	J1=     0.000 deg,	J2=   180.000 deg
};
P[172]{
   GP1:
	UF : 1, UT : 1,		CONFIG : 'N U T, 0, 0, 0',
	X =  2112.025  mm,	Y =   402.590  mm,	Z =  1192.449  mm,
	W =      .016 deg,	P =     -.045 deg,	R =   -23.885 deg
   GP2:
	UF : 1, UT : 1,
	J1=   135.000 deg,	J2=     0.000 deg
};
P[173]{
   GP1:
	UF : 1, UT : 1,		CONFIG : 'N U T, 0, 0, 0',
	X =  2111.810  mm,	Y =    14.647  mm,	Z =  1192.450  mm,
	W =      .016 deg,	P =     -.045 deg,	R =   -23.885 deg
   GP2:
	UF : 1, UT : 1,
	J1=   135.000 deg,	J2=     0.000 deg
};
P[174]{
   GP1:
	UF : 1, UT : 1,		CONFIG : 'N U T, 0, 0, 0',
	X =  1543.269  mm,	Y =  -478.741  mm,	Z =    98.416  mm,
	W =   -16.138 deg,	P =    42.751 deg,	R =   168.873 deg
   GP2:
	UF : 1, UT : 1,
	J1=     0.000 deg,	J2=   180.000 deg
};
P[175]{
   GP1:
	UF : 1, UT : 1,		CONFIG : 'N U T, 0, 0, 0',
	X =  1494.684  mm,	Y =    -9.285  mm,	Z =   211.201  mm,
	W =    -1.993 deg,	P =    44.965 deg,	R =   177.180 deg
   GP2:
	UF : 1, UT : 1,
	J1=     0.000 deg,	J2=   180.000 deg
};
P[176]{
   GP1:
	UF : 1, UT : 1,		CONFIG : 'N U T, 0, 0, 0',
	X =  2128.997  mm,	Y =  -645.877  mm,	Z =  1179.040  mm,
	W =     -.110 deg,	P =     -.657 deg,	R =   -23.879 deg
   GP2:
	UF : 1, UT : 1,
	J1=   135.000 deg,	J2=     0.000 deg
};
P[177]{
   GP1:
	UF : 1, UT : 1,		CONFIG : 'N U T, 0, 0, 0',
	X =  2128.776  mm,	Y =  -455.457  mm,	Z =  1177.054  mm,
	W =     -.064 deg,	P =    -1.106 deg,	R =   -23.872 deg
   GP2:
	UF : 1, UT : 1,
	J1=   135.000 deg,	J2=     0.000 deg
};
P[178]{
   GP1:
	UF : 1, UT : 1,		CONFIG : 'N U T, 0, 0, 0',
	X =  1534.968  mm,	Y =  -398.034  mm,	Z =    84.062  mm,
	W =     -.043 deg,	P =    44.368 deg,	R =   176.047 deg
   GP2:
	UF : 1, UT : 1,
	J1=     0.000 deg,	J2=   180.000 deg
};
P[179]{
   GP1:
	UF : 1, UT : 1,		CONFIG : 'N U T, 0, 0, 0',
	X =  1493.431  mm,	Y =   363.490  mm,	Z =   189.000  mm,
	W =   -16.664 deg,	P =    42.430 deg,	R =   156.075 deg
   GP2:
	UF : 1, UT : 1,
	J1=     0.000 deg,	J2=   180.000 deg
};
P[180]{
   GP1:
	UF : 1, UT : 1,		CONFIG : 'N U T, 0, 0, 0',
	X =  2129.638  mm,	Y =  -446.131  mm,	Z =  1180.944  mm,
	W =     3.415 deg,	P =     -.816 deg,	R =   -23.974 deg
   GP2:
	UF : 1, UT : 1,
	J1=   135.000 deg,	J2=     0.000 deg
};
P[181]{
   GP1:
	UF : 1, UT : 1,		CONFIG : 'N U T, 0, 0, 0',
	X =  2353.698  mm,	Y =   399.991  mm,	Z =   291.072  mm,
	W =    43.149 deg,	P =    14.488 deg,	R =   -37.828 deg
   GP2:
	UF : 1, UT : 1,
	J1=      .000 deg,	J2=   180.000 deg
};
P[182]{
   GP1:
	UF : 1, UT : 1,		CONFIG : 'N U T, 0, 0, 0',
	X =  1481.802  mm,	Y =    -4.268  mm,	Z =   197.574  mm,
	W =    -1.993 deg,	P =    44.965 deg,	R =   177.180 deg
   GP2:
	UF : 1, UT : 1,
	J1=     0.000 deg,	J2=   180.000 deg
};
P[183]{
   GP1:
	UF : 1, UT : 1,		CONFIG : 'N U T, 0, 0, 0',
	X =  1481.802  mm,	Y =   612.875  mm,	Z =   197.574  mm,
	W =   -40.373 deg,	P =    21.850 deg,	R =   111.598 deg
   GP2:
	UF : 1, UT : 1,
	J1=     0.000 deg,	J2=   180.000 deg
};
P[184]{
   GP1:
	UF : 1, UT : 1,		CONFIG : 'N U T, 0, 0, 0',
	X =  2345.067  mm,	Y =   409.224  mm,	Z =   281.500  mm,
	W =    43.108 deg,	P =    14.444 deg,	R =   -17.326 deg
   GP2:
	UF : 1, UT : 1,
	J1=     0.000 deg,	J2=   180.000 deg
};
P[185]{
   GP1:
	UF : 1, UT : 1,		CONFIG : 'N U T, 0, 0, 0',
	X =  2306.742  mm,	Y =   406.911  mm,	Z =   281.490  mm,
	W =    43.110 deg,	P =    14.442 deg,	R =   -17.330 deg
   GP2:
	UF : 1, UT : 1,
	J1=     0.000 deg,	J2=   180.000 deg
};
P[186]{
   GP1:
	UF : 1, UT : 1,		CONFIG : 'N U T, 0, 0, -1',
	X =  1406.501  mm,	Y =   510.995  mm,	Z =   296.764  mm,
	W =   -40.802 deg,	P =    20.911 deg,	R =   112.463 deg
   GP2:
	UF : 1, UT : 1,
	J1=     0.000 deg,	J2=   180.000 deg
};
P[187]{
   GP1:
	UF : 1, UT : 1,		CONFIG : 'N U T, 0, 0, 0',
	X =  1226.008  mm,	Y =   -21.205  mm,	Z =   297.416  mm,
	W =      .340 deg,	P =    45.409 deg,	R =    12.184 deg
   GP2:
	UF : 1, UT : 1,
	J1=     0.000 deg,	J2=   180.000 deg
};
P[188]{
   GP1:
	UF : 1, UT : 1,		CONFIG : 'N U T, 0, 0, 0',
	X =  2197.405  mm,	Y =   -25.809  mm,	Z =  -200.004  mm,
	W =     -.223 deg,	P =     -.454 deg,	R =     -.269 deg
   GP2:
	UF : 1, UT : 1,
	J1=    45.206 deg,	J2=   180.000 deg
};
P[189]{
   GP1:
	UF : 1, UT : 1,		CONFIG : 'N U T, 0, 0, 0',
	X =  2305.896  mm,	Y =   -25.032  mm,	Z =  -270.188  mm,
	W =      .477 deg,	P =    12.556 deg,	R =     -.810 deg
   GP2:
	UF : 1, UT : 1,
	J1=    45.206 deg,	J2=   180.000 deg
};
P[190]{
   GP1:
	UF : 1, UT : 1,		CONFIG : 'N U T, 0, 0, 0',
	X =  2290.712  mm,	Y =   409.911  mm,	Z =   281.500  mm,
	W =    43.107 deg,	P =    14.443 deg,	R =    14.426 deg
   GP2:
	UF : 1, UT : 1,
	J1=     0.000 deg,	J2=   180.000 deg
};
P[191]{
   GP1:
	UF : 1, UT : 1,		CONFIG : 'N U T, 0, 0, 0',
	X =  2361.728  mm,	Y =  -412.684  mm,	Z =   283.675  mm,
	W =   -31.226 deg,	P =   -24.163 deg,	R =    -2.589 deg
   GP2:
	UF : 1, UT : 1,
	J1=     0.000 deg,	J2=   180.000 deg
};
P[192]{
   GP1:
	UF : 1, UT : 1,		CONFIG : 'N U T, 0, 0, 0',
	X =  2327.653  mm,	Y =   -25.077  mm,	Z =  -148.093  mm,
	W =      .476 deg,	P =    12.559 deg,	R =     -.810 deg
   GP2:
	UF : 1, UT : 1,
	J1=    45.206 deg,	J2=   180.000 deg
};
P[193]{
   GP1:
	UF : 1, UT : 1,		CONFIG : 'N U T, 0, 0, 0',
	X =  1727.799  mm,	Y =   -46.845  mm,	Z =   458.542  mm,
	W =     2.935 deg,	P =   -34.514 deg,	R =   -11.373 deg
   GP2:
	UF : 1, UT : 1,
	J1=     0.000 deg,	J2=   180.000 deg
};
P[194]{
   GP1:
	UF : 1, UT : 1,		CONFIG : 'N U T, 0, 0, 0',
	X =  2344.238  mm,	Y =  -414.136  mm,	Z =   281.331  mm,
	W =   -33.506 deg,	P =   -24.171 deg,	R =   -30.020 deg
   GP2:
	UF : 1, UT : 1,
	J1=     0.000 deg,	J2=   180.000 deg
};
P[195]{
   GP1:
	UF : 1, UT : 1,		CONFIG : 'N U T, 0, 0, 0',
	X =  2303.808  mm,	Y =  -413.308  mm,	Z =   281.330  mm,
	W =   -33.506 deg,	P =   -24.171 deg,	R =   -30.020 deg
   GP2:
	UF : 1, UT : 1,
	J1=     0.000 deg,	J2=   180.000 deg
};
P[196]{
   GP1:
	UF : 1, UT : 1,		CONFIG : 'N U T, 0, 0, 0',
	X =  1670.118  mm,	Y =  -166.484  mm,	Z =   -15.328  mm,
	W =     1.674 deg,	P =   -29.607 deg,	R =   -12.085 deg
   GP2:
	UF : 1, UT : 1,
	J1=     0.000 deg,	J2=   180.000 deg
};
P[197]{
   GP1:
	UF : 1, UT : 1,		CONFIG : 'N U T, 0, 0, 0',
	X =  2284.901  mm,	Y =  -412.985  mm,	Z =   282.798  mm,
	W =   -33.505 deg,	P =   -24.171 deg,	R =   -60.790 deg
   GP2:
	UF : 1, UT : 1,
	J1=     0.000 deg,	J2=   180.000 deg
};
P[198]{
   GP1:
	UF : 1, UT : 1,		CONFIG : 'N U T, 0, 0, 0',
	X =  2368.954  mm,	Y =  -246.180  mm,	Z =  -185.021  mm,
	W =    35.524 deg,	P =    28.328 deg,	R =  -122.465 deg
   GP2:
	UF : 1, UT : 1,
	J1=      .000 deg,	J2=   180.000 deg
};
P[199]{
   GP1:
	UF : 1, UT : 1,		CONFIG : 'N U T, 0, 0, 0',
	X =  1667.363  mm,	Y =  -120.483  mm,	Z =     2.410  mm,
	W =     6.134 deg,	P =   -28.692 deg,	R =   -14.256 deg
   GP2:
	UF : 1, UT : 1,
	J1=     0.000 deg,	J2=   180.000 deg
};
P[200]{
   GP1:
	UF : 1, UT : 1,		CONFIG : 'N U T, 0, 0, 0',
	X =  1526.901  mm,	Y =   -72.453  mm,	Z =   656.445  mm,
	W =   -14.352 deg,	P =    -5.632 deg,	R =   -30.177 deg
   GP2:
	UF : 1, UT : 1,
	J1=     0.000 deg,	J2=   180.000 deg
};
P[201]{
   GP1:
	UF : 1, UT : 1,		CONFIG : 'N U T, 0, 0, 0',
	X =   918.616  mm,	Y =  -238.769  mm,	Z =   572.023  mm,
	W =    44.545 deg,	P =     7.177 deg,	R =    -7.219 deg
   GP2:
	UF : 1, UT : 1,
	J1=    80.000 deg,	J2=    90.000 deg
};
P[202]{
   GP1:
	UF : 1, UT : 1,		CONFIG : 'N U T, 0, 0, 0',
	X =  1548.492  mm,	Y = -1079.480  mm,	Z =  1677.351  mm,
	W =   -38.101 deg,	P =   -29.846 deg,	R =   -22.090 deg
   GP2:
	UF : 1, UT : 1,
	J1=   180.000 deg,	J2=   -90.000 deg
};
P[203]{
   GP1:
	UF : 1, UT : 1,		CONFIG : 'N U T, 0, 0, 0',
	X =  2472.617  mm,	Y =   -96.769  mm,	Z =    57.023  mm,
	W =    44.545 deg,	P =     7.177 deg,	R =    -7.219 deg
   GP2:
	UF : 1, UT : 1,
	J1=    80.000 deg,	J2=    90.000 deg
};
P[204]{
   GP1:
	UF : 1, UT : 1,		CONFIG : 'N U T, 0, 0, 0',
	X =  2434.636  mm,	Y =    22.422  mm,	Z =     9.532  mm,
	W =    44.545 deg,	P =     7.177 deg,	R =     8.203 deg
   GP2:
	UF : 1, UT : 1,
	J1=    80.000 deg,	J2=    90.000 deg
};
P[205]{
   GP1:
	UF : 1, UT : 1,		CONFIG : 'N U T, 0, 0, 0',
	X =  2368.508  mm,	Y =  -153.263  mm,	Z =  -185.665  mm,
	W =    29.649 deg,	P =    34.164 deg,	R =  -132.677 deg
   GP2:
	UF : 1, UT : 1,
	J1=      .000 deg,	J2=   180.000 deg
};
P[206]{
   GP1:
	UF : 1, UT : 1,		CONFIG : 'N U T, 0, 0, -1',
	X =  2368.281  mm,	Y =   236.535  mm,	Z =  -188.580  mm,
	W =    -9.595 deg,	P =    42.288 deg,	R =   171.259 deg
   GP2:
	UF : 1, UT : 1,
	J1=      .000 deg,	J2=   180.000 deg
};
P[207]{
   GP1:
	UF : 1, UT : 1,		CONFIG : 'N U T, 0, 0, 0',
	X =  2432.636  mm,	Y =    17.422  mm,	Z =     9.532  mm,
	W =    44.545 deg,	P =     7.177 deg,	R =     8.203 deg
   GP2:
	UF : 1, UT : 1,
	J1=    80.000 deg,	J2=    90.000 deg
};
P[208]{
   GP1:
	UF : 1, UT : 1,		CONFIG : 'N U T, 0, 0, 0',
	X =  2480.777  mm,	Y =    17.423  mm,	Z =     9.532  mm,
	W =    44.545 deg,	P =     7.177 deg,	R =    58.110 deg
   GP2:
	UF : 1, UT : 1,
	J1=    80.000 deg,	J2=    90.000 deg
};
P[209]{
   GP1:
	UF : 1, UT : 1,		CONFIG : 'N U T, 0, 0, 0',
	X =  1635.388  mm,	Y =  -650.992  mm,	Z =     9.397  mm,
	W =   -29.288 deg,	P =    36.027 deg,	R =   140.467 deg
   GP2:
	UF : 1, UT : 1,
	J1=     0.000 deg,	J2=   180.000 deg
};
P[210]{
   GP1:
	UF : 1, UT : 1,		CONFIG : 'N U T, 0, 0, 0',
	X =  1636.073  mm,	Y =  -463.277  mm,	Z =     9.397  mm,
	W =   -29.288 deg,	P =    36.027 deg,	R =   140.467 deg
   GP2:
	UF : 1, UT : 1,
	J1=     0.000 deg,	J2=   180.000 deg
};
P[211]{
   GP1:
	UF : 1, UT : 1,		CONFIG : 'N U T, 0, 0, 0',
	X =  2482.777  mm,	Y =    35.280  mm,	Z =     9.532  mm,
	W =    44.545 deg,	P =     7.177 deg,	R =    63.931 deg
   GP2:
	UF : 1, UT : 1,
	J1=    80.000 deg,	J2=    90.000 deg
};
P[212]{
   GP1:
	UF : 1, UT : 1,		CONFIG : 'N U T, 0, 0, 0',
	X =  2482.776  mm,	Y =  -110.577  mm,	Z =     9.532  mm,
	W =    44.545 deg,	P =     7.177 deg,	R =    58.110 deg
   GP2:
	UF : 1, UT : 1,
	J1=    80.000 deg,	J2=    90.000 deg
};
P[213]{
   GP1:
	UF : 1, UT : 1,		CONFIG : 'N U T, 0, 0, 0',
	X =  1737.776  mm,	Y =  -110.577  mm,	Z =   268.532  mm,
	W =    44.545 deg,	P =     7.177 deg,	R =   -14.147 deg
   GP2:
	UF : 1, UT : 1,
	J1=    80.000 deg,	J2=    90.000 deg
};
P[214]{
   GP1:
	UF : 1, UT : 1,		CONFIG : 'N U T, 0, 0, 0',
	X =  1737.776  mm,	Y =  -154.258  mm,	Z =    41.532  mm,
	W =     6.301 deg,	P =    44.648 deg,	R =   -72.376 deg
   GP2:
	UF : 1, UT : 1,
	J1=    90.000 deg,	J2=    90.000 deg
};
P[215]{
   GP1:
	UF : 1, UT : 1,		CONFIG : 'N U T, 0, 0, 0',
	X =  1633.816  mm,	Y =  -450.420  mm,	Z =     9.396  mm,
	W =   -29.288 deg,	P =    36.027 deg,	R =   154.755 deg
   GP2:
	UF : 1, UT : 1,
	J1=     0.000 deg,	J2=   180.000 deg
};
P[216]{
   GP1:
	UF : 1, UT : 1,		CONFIG : 'N U T, 0, 0, -1',
	X =  1613.596  mm,	Y =    -4.272  mm,	Z =     8.234  mm,
	W =     -.047 deg,	P =    44.367 deg,	R =   176.045 deg
   GP2:
	UF : 1, UT : 1,
	J1=     0.000 deg,	J2=   180.000 deg
};
P[217]{
   GP1:
	UF : 1, UT : 1,		CONFIG : 'N U T, 0, 0, 0',
	X =  1612.710  mm,	Y =  -390.605  mm,	Z =     8.243  mm,
	W =     -.043 deg,	P =    44.368 deg,	R =   176.047 deg
   GP2:
	UF : 1, UT : 1,
	J1=     0.000 deg,	J2=   180.000 deg
};
P[218]{
   GP1:
	UF : 1, UT : 1,		CONFIG : 'N U T, 0, 0, -1',
	X =  1614.350  mm,	Y =   382.409  mm,	Z =     8.443  mm,
	W =   -16.664 deg,	P =    42.430 deg,	R =   156.075 deg
   GP2:
	UF : 1, UT : 1,
	J1=     0.000 deg,	J2=   180.000 deg
};
P[219]{
   GP1:
	UF : 1, UT : 1,		CONFIG : 'N U T, 0, 0, 0',
	X =  1948.457  mm,	Y =  -171.292  mm,	Z =    74.447  mm,
	W =    25.119 deg,	P =    38.698 deg,	R =   -79.648 deg
   GP2:
	UF : 1, UT : 1,
	J1=    90.000 deg,	J2=    90.000 deg
};
P[220]{
   GP1:
	UF : 1, UT : 1,		CONFIG : 'N U T, 0, 0, 0',
	X =  2211.458  mm,	Y =   -28.292  mm,	Z =    74.447  mm,
	W =    40.079 deg,	P =    22.554 deg,	R =   -29.245 deg
   GP2:
	UF : 1, UT : 1,
	J1=    90.000 deg,	J2=    90.000 deg
};
P[221]{
   GP1:
	UF : 1, UT : 1,		CONFIG : 'N U T, 0, 0, -1',
	X =  1613.608  mm,	Y =    -1.137  mm,	Z =     8.022  mm,
	W =      .311 deg,	P =    44.999 deg,	R =   176.092 deg
   GP2:
	UF : 1, UT : 1,
	J1=     0.000 deg,	J2=   180.000 deg
};
P[222]{
   GP1:
	UF : 1, UT : 1,		CONFIG : 'N U T, 0, 0, -1',
	X =  1639.839  mm,	Y =   639.136  mm,	Z =     5.114  mm,
	W =   -40.728 deg,	P =    21.070 deg,	R =   110.622 deg
   GP2:
	UF : 1, UT : 1,
	J1=     0.000 deg,	J2=   180.000 deg
};
P[223]{
   GP1:
	UF : 1, UT : 1,		CONFIG : 'N U T, 0, 0, 0',
	X =  2211.458  mm,	Y =   -28.292  mm,	Z =    74.447  mm,
	W =    40.079 deg,	P =    22.554 deg,	R =   -29.245 deg
   GP2:
	UF : 1, UT : 1,
	J1=    90.000 deg,	J2=    90.000 deg
};
P[224]{
   GP1:
	UF : 1, UT : 1,		CONFIG : 'N U T, 0, 0, -1',
	X =  1639.963  mm,	Y =   451.620  mm,	Z =     4.298  mm,
	W =   -40.729 deg,	P =    21.083 deg,	R =   110.640 deg
   GP2:
	UF : 1, UT : 1,
	J1=     0.000 deg,	J2=   180.000 deg
};
P[225]{
   GP1:
	UF : 1, UT : 1,		CONFIG : 'N U T, 0, 0, -1',
	X =  1635.945  mm,	Y =   445.191  mm,	Z =     7.824  mm,
	W =   -40.728 deg,	P =    21.070 deg,	R =    97.581 deg
   GP2:
	UF : 1, UT : 1,
	J1=     0.000 deg,	J2=   180.000 deg
};
P[226]{
   GP1:
	UF : 1, UT : 1,		CONFIG : 'N U T, 0, 0, 0',
	X =  2205.310  mm,	Y =   -25.576  mm,	Z =    66.898  mm,
	W =    38.911 deg,	P =    24.669 deg,	R =   -27.342 deg
   GP2:
	UF : 1, UT : 1,
	J1=    90.000 deg,	J2=    90.000 deg
};
P[227]{
   GP1:
	UF : 1, UT : 1,		CONFIG : 'N U T, 0, 0, 0',
	X =  2091.876  mm,	Y =   -25.576  mm,	Z =    66.898  mm,
	W =    38.911 deg,	P =    24.669 deg,	R =   -27.342 deg
   GP2:
	UF : 1, UT : 1,
	J1=    90.000 deg,	J2=    90.000 deg
};
P[228]{
   GP1:
	UF : 1, UT : 1,		CONFIG : 'N U T, 0, 0, 0',
	X =  2293.114  mm,	Y =   -80.867  mm,	Z =  -319.665  mm,
	W =     -.121 deg,	P =    25.433 deg,	R =      .191 deg
   GP2:
	UF : 1, UT : 1,
	J1=    45.000 deg,	J2=   180.000 deg
};
P[229]{
   GP1:
	UF : 1, UT : 1,		CONFIG : 'N U T, 0, 0, 0',
	X =  2294.205  mm,	Y =  -160.262  mm,	Z =  -320.161  mm,
	W =    -3.243 deg,	P =    25.371 deg,	R =    16.072 deg
   GP2:
	UF : 1, UT : 1,
	J1=    45.000 deg,	J2=   180.000 deg
};
P[230]{
   GP1:
	UF : 1, UT : 1,		CONFIG : 'N U T, 0, 0, 0',
	X =  2037.608  mm,	Y =   -74.366  mm,	Z =   106.547  mm,
	W =    38.909 deg,	P =    24.669 deg,	R =   -38.380 deg
   GP2:
	UF : 1, UT : 1,
	J1=    90.000 deg,	J2=    90.000 deg
};
P[231]{
   GP1:
	UF : 1, UT : 1,		CONFIG : 'N U T, 0, 0, 0',
	X =  1708.547  mm,	Y =  -153.366  mm,	Z =    49.547  mm,
	W =    38.909 deg,	P =    24.669 deg,	R =    46.020 deg
   GP2:
	UF : 1, UT : 1,
	J1=    90.000 deg,	J2=    90.000 deg
};
P[232]{
   GP1:
	UF : 1, UT : 1,		CONFIG : 'N U T, 0, 0, 0',
	X =  1683.626  mm,	Y =   -81.655  mm,	Z =   -53.149  mm,
	W =    10.416 deg,	P =   -27.285 deg,	R =   -21.847 deg
   GP2:
	UF : 1, UT : 1,
	J1=     0.000 deg,	J2=   180.000 deg
};
P[233]{
   GP1:
	UF : 1, UT : 1,		CONFIG : 'N U T, 0, 0, 0',
	X =  1683.155  mm,	Y =  -106.369  mm,	Z =   -53.149  mm,
	W =    10.416 deg,	P =   -27.285 deg,	R =   -21.847 deg
   GP2:
	UF : 1, UT : 1,
	J1=     0.000 deg,	J2=   180.000 deg
};
P[234]{
   GP1:
	UF : 1, UT : 1,		CONFIG : 'N U T, 0, 0, 0',
	X =  1744.400  mm,	Y =  -130.049  mm,	Z =    76.607  mm,
	W =    33.797 deg,	P =    31.690 deg,	R =    32.974 deg
   GP2:
	UF : 1, UT : 1,
	J1=    90.000 deg,	J2=    90.000 deg
};
P[235]{
   GP1:
	UF : 1, UT : 1,		CONFIG : 'N U T, 0, 0, 0',
	X =  1890.431  mm,	Y =   -61.192  mm,	Z =   115.273  mm,
	W =    39.113 deg,	P =    33.534 deg,	R =   -57.069 deg
   GP2:
	UF : 1, UT : 1,
	J1=    90.000 deg,	J2=    90.000 deg
};
P[236]{
   GP1:
	UF : 1, UT : 1,		CONFIG : 'N U T, 0, 0, 0',
	X =  1684.182  mm,	Y =  -159.370  mm,	Z =   -53.149  mm,
	W =    12.300 deg,	P =   -26.597 deg,	R =   -22.701 deg
   GP2:
	UF : 1, UT : 1,
	J1=     0.000 deg,	J2=   180.000 deg
};
P[237]{
   GP1:
	UF : 1, UT : 1,		CONFIG : 'N U T, 0, 0, 0',
	X =  1825.520  mm,	Y =      .488  mm,	Z =    92.358  mm,
	W =    44.280 deg,	P =    22.416 deg,	R =   -25.152 deg
   GP2:
	UF : 1, UT : 1,
	J1=    89.996 deg,	J2=    90.000 deg
};
P[238]{
   GP1:
	UF : 1, UT : 1,		CONFIG : 'N U T, 0, 0, 0',
	X =  1684.208  mm,	Y =  -131.065  mm,	Z =   -53.167  mm,
	W =    12.285 deg,	P =   -26.598 deg,	R =   -22.689 deg
   GP2:
	UF : 1, UT : 1,
	J1=     0.000 deg,	J2=   180.000 deg
};
P[239]{
   GP1:
	UF : 1, UT : 1,		CONFIG : 'N U T, 0, 0, 0',
	X =  2450.528  mm,	Y =    67.264  mm,	Z =   -29.881  mm,
	W =    43.929 deg,	P =   -14.757 deg,	R =    26.953 deg
   GP2:
	UF : 1, UT : 1,
	J1=    80.000 deg,	J2=    90.000 deg
};
P[240]{
   GP1:
	UF : 1, UT : 1,		CONFIG : 'N U T, 0, 0, 0',
	X =  2391.317  mm,	Y =    67.003  mm,	Z =   -18.123  mm,
	W =    47.953 deg,	P =      .226 deg,	R =    27.045 deg
   GP2:
	UF : 1, UT : 1,
	J1=    80.000 deg,	J2=    90.000 deg
};
P[241]{
   GP1:
	UF : 1, UT : 1,		CONFIG : 'N U T, 0, 0, 0',
	X =  2378.694  mm,	Y =    65.889  mm,	Z =   -21.684  mm,
	W =    47.614 deg,	P =     2.717 deg,	R =    43.711 deg
   GP2:
	UF : 1, UT : 1,
	J1=    80.000 deg,	J2=    90.000 deg
};
P[242]{
   GP1:
	UF : 1, UT : 1,		CONFIG : 'N U T, 0, 0, 0',
	X =  1722.530  mm,	Y =   -86.452  mm,	Z =   134.799  mm,
	W =    51.320 deg,	P =    22.528 deg,	R =    10.143 deg
   GP2:
	UF : 1, UT : 1,
	J1=    89.999 deg,	J2=    90.000 deg
};
P[243]{
   GP1:
	UF : 1, UT : 1,		CONFIG : 'N U T, 0, 0, 0',
	X =  1245.855  mm,	Y =  -163.909  mm,	Z =   181.900  mm,
	W =     8.587 deg,	P =    44.350 deg,	R =   -94.561 deg
   GP2:
	UF : 1, UT : 1,
	J1=    90.000 deg,	J2=    90.000 deg
};
P[244]{
   GP1:
	UF : 1, UT : 1,		CONFIG : 'N U T, 0, 0, 0',
	X =  1175.771  mm,	Y =   480.202  mm,	Z =   147.755  mm,
	W =     5.148 deg,	P =    45.783 deg,	R =    38.993 deg
   GP2:
	UF : 1, UT : 1,
	J1=    90.000 deg,	J2=    90.000 deg
};
P[245]{
   GP1:
	UF : 1, UT : 1,		CONFIG : 'N U T, 0, 0, 0',
	X =  2149.855  mm,	Y =   157.091  mm,	Z =   181.900  mm,
	W =   -44.543 deg,	P =     7.216 deg,	R =     5.945 deg
   GP2:
	UF : 1, UT : 1,
	J1=    90.000 deg,	J2=    90.000 deg
};
P[246]{
   GP1:
	UF : 1, UT : 1,		CONFIG : 'N U T, 0, 0, 0',
	X =  2375.455  mm,	Y =    62.722  mm,	Z =   -19.359  mm,
	W =    52.026 deg,	P =    21.224 deg,	R =    45.474 deg
   GP2:
	UF : 1, UT : 1,
	J1=    80.000 deg,	J2=    90.000 deg
};
P[247]{
   GP1:
	UF : 1, UT : 1,		CONFIG : 'N U T, 0, 0, 0',
	X =  2372.087  mm,	Y =    46.546  mm,	Z =   -20.713  mm,
	W =    52.025 deg,	P =    21.226 deg,	R =    71.331 deg
   GP2:
	UF : 1, UT : 1,
	J1=    80.000 deg,	J2=    90.000 deg
};
P[248]{
   GP1:
	UF : 1, UT : 1,		CONFIG : 'N U T, 0, 0, 0',
	X =  2142.216  mm,	Y =   113.042  mm,	Z =    61.147  mm,
	W =   -44.622 deg,	P =     6.557 deg,	R =     6.600 deg
   GP2:
	UF : 1, UT : 1,
	J1=    90.000 deg,	J2=    90.000 deg
};
P[249]{
   GP1:
	UF : 1, UT : 1,		CONFIG : 'N U T, 0, 0, 0',
	X =  2373.771  mm,	Y =     9.115  mm,	Z =   -18.796  mm,
	W =    52.027 deg,	P =    21.227 deg,	R =    74.733 deg
   GP2:
	UF : 1, UT : 1,
	J1=    80.000 deg,	J2=    90.000 deg
};
P[250]{
   GP1:
	UF : 1, UT : 1,		CONFIG : 'N U T, 0, 0, 0',
	X =  2372.598  mm,	Y =    -5.392  mm,	Z =   -19.166  mm,
	W =    52.021 deg,	P =    21.222 deg,	R =    96.043 deg
   GP2:
	UF : 1, UT : 1,
	J1=    80.000 deg,	J2=    90.000 deg
};
P[251]{
   GP1:
	UF : 1, UT : 1,		CONFIG : 'N U T, 0, 0, 0',
	X =  2213.194  mm,	Y =   163.254  mm,	Z =   103.953  mm,
	W =   -44.622 deg,	P =     6.557 deg,	R =     6.600 deg
   GP2:
	UF : 1, UT : 1,
	J1=    90.000 deg,	J2=    90.000 deg
};
P[252]{
   GP1:
	UF : 1, UT : 1,		CONFIG : 'N U T, 0, 0, 0',
	X =  1974.194  mm,	Y =   163.254  mm,	Z =   103.953  mm,
	W =   -44.622 deg,	P =     6.557 deg,	R =     6.600 deg
   GP2:
	UF : 1, UT : 1,
	J1=    90.000 deg,	J2=    90.000 deg
};
P[253]{
   GP1:
	UF : 1, UT : 1,		CONFIG : 'N U T, 0, 0, 0',
	X =  1672.125  mm,	Y =   -94.766  mm,	Z =   -11.860  mm,
	W =      .944 deg,	P =    45.049 deg,	R =   -47.839 deg
   GP2:
	UF : 1, UT : 1,
	J1=    90.000 deg,	J2=    90.000 deg
};
P[254]{
   GP1:
	UF : 1, UT : 1,		CONFIG : 'N U T, 0, 0, 0',
	X =  1703.433  mm,	Y =   -94.616  mm,	Z =   -13.144  mm,
	W =      .965 deg,	P =    44.871 deg,	R =   -92.736 deg
   GP2:
	UF : 1, UT : 1,
	J1=    90.000 deg,	J2=    90.000 deg
};
P[255]{
   GP1:
	UF : 1, UT : 1,		CONFIG : 'N U T, 0, 0, 0',
	X =  1982.874  mm,	Y =   -97.216  mm,	Z =   -12.026  mm,
	W =      .937 deg,	P =    45.000 deg,	R =   -93.403 deg
   GP2:
	UF : 1, UT : 1,
	J1=    90.000 deg,	J2=    90.000 deg
};
P[256]{
   GP1:
	UF : 1, UT : 1,		CONFIG : 'N U T, 0, 0, 0',
	X =  2011.831  mm,	Y =   189.641  mm,	Z =   186.534  mm,
	W =   -48.207 deg,	P =    -3.724 deg,	R =    27.867 deg
   GP2:
	UF : 1, UT : 1,
	J1=    90.000 deg,	J2=    90.000 deg
};
P[257]{
   GP1:
	UF : 1, UT : 1,		CONFIG : 'N U T, 0, 0, 0',
	X =  2155.758  mm,	Y =    17.641  mm,	Z =    61.534  mm,
	W =   -48.207 deg,	P =    -3.724 deg,	R =   -86.423 deg
   GP2:
	UF : 1, UT : 1,
	J1=    90.000 deg,	J2=   100.000 deg
};
P[258]{
   GP1:
	UF : 1, UT : 1,		CONFIG : 'N U T, 0, 0, 0',
	X =  1996.444  mm,	Y =   -96.787  mm,	Z =   -12.026  mm,
	W =      .937 deg,	P =    45.000 deg,	R =  -125.609 deg
   GP2:
	UF : 1, UT : 1,
	J1=    90.000 deg,	J2=    90.000 deg
};
P[259]{
   GP1:
	UF : 1, UT : 1,		CONFIG : 'N U T, 0, 0, 0',
	X =  2228.536  mm,	Y =    43.219  mm,	Z =     3.885  mm,
	W =    38.936 deg,	P =    24.695 deg,	R =   -29.101 deg
   GP2:
	UF : 1, UT : 1,
	J1=    89.999 deg,	J2=    90.000 deg
};
P[260]{
   GP1:
	UF : 1, UT : 1,		CONFIG : 'N U T, 0, 0, 0',
	X =  2155.758  mm,	Y =    17.641  mm,	Z =   102.048  mm,
	W =   -48.207 deg,	P =    -3.724 deg,	R =   -86.423 deg
   GP2:
	UF : 1, UT : 1,
	J1=    90.000 deg,	J2=   100.000 deg
};
P[261]{
   GP1:
	UF : 1, UT : 1,		CONFIG : 'N U T, 0, 0, 0',
	X =  2233.490  mm,	Y =   120.495  mm,	Z =   200.684  mm,
	W =   -48.207 deg,	P =    -3.724 deg,	R =   -26.585 deg
   GP2:
	UF : 1, UT : 1,
	J1=    90.000 deg,	J2=   100.000 deg
};
P[262]{
   GP1:
	UF : 1, UT : 1,		CONFIG : 'N U T, 0, 0, 0',
	X =  1849.669  mm,	Y =   238.423  mm,	Z =   211.646  mm,
	W =    32.273 deg,	P =    -6.861 deg,	R =   -73.357 deg
   GP2:
	UF : 1, UT : 1,
	J1=    90.000 deg,	J2=    90.000 deg
};
P[263]{
   GP1:
	UF : 1, UT : 1,		CONFIG : 'N U T, 0, 0, 0',
	X =  1949.669  mm,	Y =   136.423  mm,	Z =    63.646  mm,
	W =    40.686 deg,	P =    -9.263 deg,	R =   -65.467 deg
   GP2:
	UF : 1, UT : 1,
	J1=    90.000 deg,	J2=    90.000 deg
};
P[264]{
   GP1:
	UF : 1, UT : 1,		CONFIG : 'N U T, 0, 0, 0',
	X =  2267.821  mm,	Y =    42.790  mm,	Z =     3.885  mm,
	W =    38.936 deg,	P =    24.695 deg,	R =   -29.101 deg
   GP2:
	UF : 1, UT : 1,
	J1=    89.999 deg,	J2=    90.000 deg
};
P[265]{
   GP1:
	UF : 1, UT : 1,		CONFIG : 'N U T, 0, 0, 0',
	X =  2154.589  mm,	Y =    41.367  mm,	Z =    -1.757  mm,
	W =    40.759 deg,	P =    25.526 deg,	R =   -26.560 deg
   GP2:
	UF : 1, UT : 1,
	J1=    90.000 deg,	J2=    90.000 deg
};
P[266]{
   GP1:
	UF : 1, UT : 1,		CONFIG : 'N U T, 0, 0, 0',
	X =  2025.245  mm,	Y =    81.350  mm,	Z =    71.561  mm,
	W =    44.528 deg,	P =     7.306 deg,	R =  -107.368 deg
   GP2:
	UF : 1, UT : 1,
	J1=    90.000 deg,	J2=    90.000 deg
};
P[267]{
   GP1:
	UF : 1, UT : 1,		CONFIG : 'N U T, 0, 0, 0',
	X =  2568.141  mm,	Y =   334.529  mm,	Z =   374.903  mm,
	W =   -11.234 deg,	P =    -5.395 deg,	R =    -6.810 deg
   GP2:
	UF : 1, UT : 1,
	J1=    90.000 deg,	J2=   135.000 deg
};
P[268]{
   GP1:
	UF : 1, UT : 1,		CONFIG : 'N U T, 0, 0, 0',
	X =  2726.458  mm,	Y =   283.351  mm,	Z =   364.849  mm,
	W =    -5.482 deg,	P =   -11.711 deg,	R =   -26.938 deg
   GP2:
	UF : 1, UT : 1,
	J1=    90.000 deg,	J2=   135.000 deg
};
P[269]{
   GP1:
	UF : 1, UT : 1,		CONFIG : 'N U T, 0, 0, 0',
	X =  2205.896  mm,	Y =    40.624  mm,	Z =    -1.591  mm,
	W =    40.756 deg,	P =    25.520 deg,	R =   -26.559 deg
   GP2:
	UF : 1, UT : 1,
	J1=    90.000 deg,	J2=    90.000 deg
};
P[270]{
   GP1:
	UF : 1, UT : 1,		CONFIG : 'N U T, 0, 0, 0',
	X =  2218.896  mm,	Y =    41.480  mm,	Z =    -1.591  mm,
	W =    40.756 deg,	P =    25.520 deg,	R =   -34.005 deg
   GP2:
	UF : 1, UT : 1,
	J1=    90.000 deg,	J2=    90.000 deg
};
P[271]{
   GP1:
	UF : 1, UT : 1,		CONFIG : 'N U T, 0, 0, 0',
	X =  2639.410  mm,	Y =   254.475  mm,	Z =   423.440  mm,
	W =    21.122 deg,	P =   -34.692 deg,	R =   -34.166 deg
   GP2:
	UF : 1, UT : 1,
	J1=    90.000 deg,	J2=   135.000 deg
};
P[272]{
   GP1:
	UF : 1, UT : 1,		CONFIG : 'N U T, 0, 0, 0',
	X =  2378.772  mm,	Y =   359.307  mm,	Z =   369.010  mm,
	W =     0.000 deg,	P =     0.000 deg,	R =     7.124 deg
   GP2:
	UF : 1, UT : 1,
	J1=    90.000 deg,	J2=   135.000 deg
};
P[273]{
   GP1:
	UF : 1, UT : 1,		CONFIG : 'N U T, 0, 0, 0',
	X =  2014.799  mm,	Y =    44.262  mm,	Z =   -12.003  mm,
	W =    38.907 deg,	P =    24.670 deg,	R =     7.094 deg
   GP2:
	UF : 1, UT : 1,
	J1=    90.000 deg,	J2=    90.000 deg
};
P[274]{
   GP1:
	UF : 1, UT : 1,		CONFIG : 'N U T, 0, 0, 0',
	X =  2041.487  mm,	Y =    43.237  mm,	Z =   -11.618  mm,
	W =    38.906 deg,	P =    24.669 deg,	R =   -20.914 deg
   GP2:
	UF : 1, UT : 1,
	J1=    90.000 deg,	J2=    90.000 deg
};
P[275]{
   GP1:
	UF : 1, UT : 1,		CONFIG : 'N U T, 0, 0, 0',
	X =  2649.319  mm,	Y =   360.965  mm,	Z =   454.435  mm,
	W =     3.160 deg,	P =   -22.165 deg,	R =   -20.317 deg
   GP2:
	UF : 1, UT : 1,
	J1=    90.000 deg,	J2=   135.000 deg
};
P[276]{
   GP1:
	UF : 1, UT : 1,		CONFIG : 'N U T, 0, 0, 0',
	X =  1814.352  mm,	Y =   347.003  mm,	Z =   560.474  mm,
	W =     3.159 deg,	P =   -22.164 deg,	R =   -20.317 deg
   GP2:
	UF : 1, UT : 1,
	J1=    90.000 deg,	J2=   135.000 deg
};
P[277]{
   GP1:
	UF : 1, UT : 1,		CONFIG : 'N U T, 0, 0, 0',
	X =  1666.319  mm,	Y =   360.964  mm,	Z =   227.632  mm,
	W =   -32.996 deg,	P =    -3.828 deg,	R =    -3.143 deg
   GP2:
	UF : 1, UT : 1,
	J1=    90.000 deg,	J2=    90.000 deg
};
P[278]{
   GP1:
	UF : 1, UT : 1,		CONFIG : 'N U T, 0, 0, 0',
	X =  1666.319  mm,	Y =   145.964  mm,	Z =    68.632  mm,
	W =   -41.776 deg,	P =    -4.262 deg,	R =    -2.522 deg
   GP2:
	UF : 1, UT : 1,
	J1=    90.000 deg,	J2=    90.000 deg
};
P[279]{
   GP1:
	UF : 1, UT : 1,		CONFIG : 'N U T, 0, 0, 0',
	X =  2098.131  mm,	Y =    40.950  mm,	Z =   -10.062  mm,
	W =    38.906 deg,	P =    24.670 deg,	R =   -27.075 deg
   GP2:
	UF : 1, UT : 1,
	J1=    90.000 deg,	J2=    90.000 deg
};
P[280]{
   GP1:
	UF : 1, UT : 1,		CONFIG : 'N U T, 0, 0, 0',
	X =  2115.487  mm,	Y =    41.450  mm,	Z =   -10.347  mm,
	W =    42.498 deg,	P =    16.438 deg,	R =   -37.568 deg
   GP2:
	UF : 1, UT : 1,
	J1=    90.000 deg,	J2=    90.000 deg
};
P[281]{
   GP1:
	UF : 1, UT : 1,		CONFIG : 'N U T, 0, 0, 0',
	X =  1668.368  mm,	Y =  -149.009  mm,	Z =   -14.846  mm,
	W =    33.806 deg,	P =    31.687 deg,	R =    49.165 deg
   GP2:
	UF : 1, UT : 1,
	J1=    90.000 deg,	J2=    90.000 deg
};
P[282]{
   GP1:
	UF : 1, UT : 1,		CONFIG : 'N U T, 0, 0, 0',
	X =  1669.978  mm,	Y =  -105.338  mm,	Z =   -13.496  mm,
	W =    33.800 deg,	P =    31.688 deg,	R =    49.167 deg
   GP2:
	UF : 1, UT : 1,
	J1=    90.000 deg,	J2=    90.000 deg
};
P[283]{
   GP1:
	UF : 1, UT : 1,		CONFIG : 'N U T, 0, 0, 0',
	X =  1671.394  mm,	Y =   -95.493  mm,	Z =   -11.426  mm,
	W =    33.800 deg,	P =    31.687 deg,	R =     5.016 deg
   GP2:
	UF : 1, UT : 1,
	J1=    90.000 deg,	J2=    90.000 deg
};
P[284]{
   GP1:
	UF : 1, UT : 1,		CONFIG : 'N U T, 0, 0, 0',
	X =  1998.286  mm,	Y =    41.338  mm,	Z =    60.142  mm,
	W =    48.322 deg,	P =    22.567 deg,	R =   -50.008 deg
   GP2:
	UF : 1, UT : 1,
	J1=    89.995 deg,	J2=    90.000 deg
};
P[285]{
   GP1:
	UF : 1, UT : 1,		CONFIG : 'N U T, 0, 0, 0',
	X =  1974.603  mm,	Y =    45.573  mm,	Z =    57.345  mm,
	W =    44.953 deg,	P =    23.885 deg,	R =   -17.360 deg
   GP2:
	UF : 1, UT : 1,
	J1=    90.000 deg,	J2=    90.000 deg
};
P[286]{
   GP1:
	UF : 1, UT : 1,		CONFIG : 'N U T, 0, 0, 0',
	X =  1820.781  mm,	Y =    45.132  mm,	Z =    58.416  mm,
	W =    44.971 deg,	P =    23.892 deg,	R =   -17.364 deg
   GP2:
	UF : 1, UT : 1,
	J1=    90.000 deg,	J2=    90.000 deg
};
P[287]{
   GP1:
	UF : 1, UT : 1,		CONFIG : 'N U T, 0, 0, 0',
	X =  1800.282  mm,	Y =    43.343  mm,	Z =    59.173  mm,
	W =    35.371 deg,	P =    21.388 deg,	R =   -19.727 deg
   GP2:
	UF : 1, UT : 1,
	J1=    90.000 deg,	J2=    90.000 deg
};
P[288]{
   GP1:
	UF : 1, UT : 1,		CONFIG : 'N U T, 0, 0, 0',
	X =  1694.138  mm,	Y =    44.082  mm,	Z =    60.326  mm,
	W =    36.317 deg,	P =    20.984 deg,	R =   -19.292 deg
   GP2:
	UF : 1, UT : 1,
	J1=    90.000 deg,	J2=    90.000 deg
};
P[289]{
   GP1:
	UF : 1, UT : 1,		CONFIG : 'N U T, 0, 0, 0',
	X =  1673.588  mm,	Y =    40.107  mm,	Z =    62.206  mm,
	W =    53.998 deg,	P =    25.339 deg,	R =    13.494 deg
   GP2:
	UF : 1, UT : 1,
	J1=    90.000 deg,	J2=    90.000 deg
};
P[290]{
   GP1:
	UF : 1, UT : 1,		CONFIG : 'N U T, 0, 0, 0',
	X =  1479.942  mm,	Y =    29.744  mm,	Z =    13.601  mm,
	W =    32.121 deg,	P =   -33.901 deg,	R =  -105.164 deg
   GP2:
	UF : 1, UT : 1,
	J1=    90.000 deg,	J2=    90.000 deg
};
P[291]{
   GP1:
	UF : 1, UT : 1,		CONFIG : 'N U T, 0, 0, 0',
	X =  1147.489  mm,	Y =  -189.741  mm,	Z =   168.329  mm,
	W =     1.315 deg,	P =    44.984 deg,	R =  -175.427 deg
   GP2:
	UF : 1, UT : 1,
	J1=    90.000 deg,	J2=    90.000 deg
};
P[292]{
   GP1:
	UF : 1, UT : 1,		CONFIG : 'N U T, 0, 0, -1',
	X =  1576.307  mm,	Y =  -183.607  mm,	Z =    68.328  mm,
	W =   -35.870 deg,	P =    29.236 deg,	R =   126.749 deg
   GP2:
	UF : 1, UT : 1,
	J1=    90.000 deg,	J2=    90.000 deg
};
P[293]{
   GP1:
	UF : 1, UT : 1,		CONFIG : 'N U T, 0, 0, 0',
	X =  2229.772  mm,	Y =    54.551  mm,	Z =     4.695  mm,
	W =   -44.618 deg,	P =     6.555 deg,	R =     6.600 deg
   GP2:
	UF : 1, UT : 1,
	J1=    90.000 deg,	J2=    90.000 deg
};
P[294]{
   GP1:
	UF : 1, UT : 1,		CONFIG : 'N U T, 0, 0, 0',
	X =  2265.914  mm,	Y =    53.909  mm,	Z =     4.695  mm,
	W =   -44.618 deg,	P =     6.555 deg,	R =     6.600 deg
   GP2:
	UF : 1, UT : 1,
	J1=    90.000 deg,	J2=    90.000 deg
};
P[295]{
   GP1:
	UF : 1, UT : 1,		CONFIG : 'N U T, 0, 0, 0',
	X =  1545.339  mm,	Y =  -110.843  mm,	Z =    97.938  mm,
	W =   -34.315 deg,	P =    31.113 deg,	R =   142.478 deg
   GP2:
	UF : 1, UT : 1,
	J1=    90.000 deg,	J2=    90.000 deg
};
P[296]{
   GP1:
	UF : 1, UT : 1,		CONFIG : 'N U T, 0, 0, 0',
	X =  1872.782  mm,	Y =  -184.571  mm,	Z =   109.509  mm,
	W =    45.016 deg,	P =     4.170 deg,	R =   -10.886 deg
   GP2:
	UF : 1, UT : 1,
	J1=    90.000 deg,	J2=    90.000 deg
};
P[297]{
   GP1:
	UF : 1, UT : 1,		CONFIG : 'N U T, 0, 0, 0',
	X =  2359.287  mm,	Y =   -66.519  mm,	Z =    63.978  mm,
	W =    44.857 deg,	P =     4.010 deg,	R =    -7.659 deg
   GP2:
	UF : 1, UT : 1,
	J1=    90.000 deg,	J2=    90.000 deg
};
P[298]{
   GP1:
	UF : 1, UT : 1,		CONFIG : 'N U T, 0, 0, 0',
	X =  2140.163  mm,	Y =    55.259  mm,	Z =    -2.456  mm,
	W =   -44.622 deg,	P =     6.557 deg,	R =     9.941 deg
   GP2:
	UF : 1, UT : 1,
	J1=    90.000 deg,	J2=    90.000 deg
};
P[299]{
   GP1:
	UF : 1, UT : 1,		CONFIG : 'N U T, 0, 0, 0',
	X =  2208.724  mm,	Y =    55.260  mm,	Z =    -1.608  mm,
	W =   -44.622 deg,	P =     6.557 deg,	R =     9.941 deg
   GP2:
	UF : 1, UT : 1,
	J1=    90.000 deg,	J2=    90.000 deg
};
P[300]{
   GP1:
	UF : 1, UT : 1,		CONFIG : 'N U T, 0, 0, 0',
	X =  2359.287  mm,	Y =   -66.519  mm,	Z =    63.978  mm,
	W =    44.857 deg,	P =     4.010 deg,	R =    -7.659 deg
   GP2:
	UF : 1, UT : 1,
	J1=    90.000 deg,	J2=    90.000 deg
};
P[301]{
   GP1:
	UF : 1, UT : 1,		CONFIG : 'N U T, 0, 0, 0',
	X =  2218.750  mm,	Y =    54.701  mm,	Z =    -1.257  mm,
	W =   -44.621 deg,	P =     6.557 deg,	R =    19.051 deg
   GP2:
	UF : 1, UT : 1,
	J1=    90.000 deg,	J2=    90.000 deg
};
P[302]{
   GP1:
	UF : 1, UT : 1,		CONFIG : 'N U T, 0, 0, 0',
	X =  1993.725  mm,	Y =    57.037  mm,	Z =   -12.551  mm,
	W =   -44.622 deg,	P =     6.557 deg,	R =    12.164 deg
   GP2:
	UF : 1, UT : 1,
	J1=    90.000 deg,	J2=    90.000 deg
};
P[303]{
   GP1:
	UF : 1, UT : 1,		CONFIG : 'N U T, 0, 0, 0',
	X =  2365.670  mm,	Y =   -13.848  mm,	Z =    70.171  mm,
	W =    46.444 deg,	P =   -12.090 deg,	R =   -13.381 deg
   GP2:
	UF : 1, UT : 1,
	J1=    90.000 deg,	J2=    90.000 deg
};
P[304]{
   GP1:
	UF : 1, UT : 1,		CONFIG : 'N U T, 0, 0, 0',
	X =  1259.286  mm,	Y =   -92.719  mm,	Z =   151.978  mm,
	W =    44.857 deg,	P =     4.010 deg,	R =    -7.659 deg
   GP2:
	UF : 1, UT : 1,
	J1=    90.000 deg,	J2=    90.000 deg
};
P[305]{
   GP1:
	UF : 1, UT : 1,		CONFIG : 'N U T, 0, 0, 0',
	X =   805.000  mm,	Y =   -92.719  mm,	Z =   623.407  mm,
	W =     2.372 deg,	P =    44.949 deg,	R =   -90.282 deg
   GP2:
	UF : 1, UT : 1,
	J1=    90.000 deg,	J2=    90.000 deg
};
P[306]{
   GP1:
	UF : 1, UT : 1,		CONFIG : 'N U T, 0, 0, 0',
	X =  1594.999  mm,	Y =  1487.710  mm,	Z =  1080.406  mm,
	W =    44.983 deg,	P =     1.340 deg,	R =    -4.979 deg
   GP2:
	UF : 0, UT : 1,
	J1=    95.000 deg,	J2=    90.000 deg
};
P[307]{
   GP1:
	UF : 1, UT : 1,		CONFIG : 'N U T, 0, 0, 0',
	X =  2536.112  mm,	Y =  1559.710  mm,	Z =  1068.235  mm,
	W =    21.780 deg,	P =   -40.404 deg,	R =   -29.962 deg
   GP2:
	UF : 0, UT : 1,
	J1=    95.000 deg,	J2=    90.000 deg
};
P[308]{
   GP1:
	UF : 1, UT : 1,		CONFIG : 'N U T, 0, 0, 0',
	X =  2669.017  mm,	Y =  1509.121  mm,	Z =  1068.235  mm,
	W =    15.908 deg,	P =   -31.536 deg,	R =   -26.500 deg
   GP2:
	UF : 0, UT : 1,
	J1=    95.000 deg,	J2=    90.000 deg
};
P[309]{
   GP1:
	UF : 1, UT : 1,		CONFIG : 'N U T, 0, 0, 0',
	X =  2099.297  mm,	Y =    56.009  mm,	Z =   -11.480  mm,
	W =   -44.622 deg,	P =     6.557 deg,	R =    12.163 deg
   GP2:
	UF : 1, UT : 1,
	J1=    90.000 deg,	J2=    90.000 deg
};
P[310]{
   GP1:
	UF : 1, UT : 1,		CONFIG : 'N U T, 0, 0, 0',
	X =  2116.377  mm,	Y =    57.272  mm,	Z =    -8.464  mm,
	W =   -44.771 deg,	P =    -5.102 deg,	R =    25.638 deg
   GP2:
	UF : 1, UT : 1,
	J1=    90.000 deg,	J2=    90.000 deg
};
P[311]{
   GP1:
	UF : 1, UT : 1,		CONFIG : 'N U T, 0, 0, 0',
	X =  2011.005  mm,	Y =    90.726  mm,	Z =    -4.431  mm,
	W =   -45.694 deg,	P =     4.659 deg,	R =   -95.347 deg
   GP2:
	UF : 1, UT : 1,
	J1=    90.000 deg,	J2=   100.000 deg
};
P[312]{
   GP1:
	UF : 1, UT : 1,		CONFIG : 'N U T, 0, 0, 0',
	X =  2009.491  mm,	Y =   -24.156  mm,	Z =   -24.443  mm,
	W =   -45.682 deg,	P =     4.633 deg,	R =   -95.341 deg
   GP2:
	UF : 1, UT : 1,
	J1=    90.000 deg,	J2=   100.000 deg
};
P[313]{
   GP1:
	UF : 1, UT : 1,		CONFIG : 'N U T, 0, 0, 0',
	X =  2074.109  mm,	Y =   104.959  mm,	Z =    -8.616  mm,
	W =    44.535 deg,	P =     7.322 deg,	R =   -84.843 deg
   GP2:
	UF : 1, UT : 1,
	J1=    90.000 deg,	J2=    90.000 deg
};
P[314]{
   GP1:
	UF : 1, UT : 1,		CONFIG : 'N U T, 0, 0, 0',
	X =  2111.582  mm,	Y =    71.102  mm,	Z =    -8.601  mm,
	W =    44.528 deg,	P =     7.306 deg,	R =   -97.132 deg
   GP2:
	UF : 1, UT : 1,
	J1=    90.000 deg,	J2=    90.000 deg
};
P[315]{
   GP1:
	UF : 1, UT : 1,		CONFIG : 'N U T, 0, 0, -1',
	X =  2124.898  mm,	Y =    57.654  mm,	Z =    -6.336  mm,
	W =    44.499 deg,	P =     7.303 deg,	R =  -123.592 deg
   GP2:
	UF : 1, UT : 1,
	J1=    90.000 deg,	J2=    90.000 deg
};
P[316]{
   GP1:
	UF : 1, UT : 1,		CONFIG : 'N U T, 0, 0, 0',
	X =  2756.445  mm,	Y =   257.823  mm,	Z =   284.445  mm,
	W =     2.460 deg,	P =     1.293 deg,	R =   -27.478 deg
   GP2:
	UF : 1, UT : 1,
	J1=    90.000 deg,	J2=   135.000 deg
};
P[317]{
   GP1:
	UF : 1, UT : 1,		CONFIG : 'N U T, 0, 0, 0',
	X =  2595.933  mm,	Y =  1529.341  mm,	Z =  1071.413  mm,
	W =    42.689 deg,	P =    16.599 deg,	R =   -42.374 deg
   GP2:
	UF : 0, UT : 1,
	J1=    95.000 deg,	J2=    90.000 deg
};
P[318]{
   GP1:
	UF : 1, UT : 1,		CONFIG : 'N U T, 0, 0, 0',
	X =  1582.432  mm,	Y =  1398.159  mm,	Z =  1444.559  mm,
	W =    11.626 deg,	P =   -25.521 deg,	R =    17.476 deg
   GP2:
	UF : 1, UT : 1,
	J1=    95.000 deg,	J2=    90.000 deg
};
P[319]{
   GP1:
	UF : 1, UT : 1,		CONFIG : 'N U T, 0, 0, 0',
	X =   918.616  mm,	Y =    -7.769  mm,	Z =  2170.023  mm,
	W =     -.010 deg,	P =   -45.000 deg,	R =     0.000 deg
   GP2:
	UF : 1, UT : 1,
	J1=   -90.000 deg,	J2=   -90.000 deg
};
P[320]{
   GP1:
	UF : 1, UT : 1,		CONFIG : 'N U T, 0, 0, 0',
	X =  1206.616  mm,	Y =   429.231  mm,	Z =  1126.817  mm,
	W =    39.016 deg,	P =   -24.484 deg,	R =   -62.925 deg
   GP2:
	UF : 1, UT : 1,
	J1=   -90.000 deg,	J2=   -90.000 deg
};
P[321]{
   GP1:
	UF : 1, UT : 1,		CONFIG : 'N U T, 0, 0, 0',
	X =  1637.790  mm,	Y =   298.510  mm,	Z =   877.535  mm,
	W =     3.496 deg,	P =   -44.892 deg,	R =    -9.391 deg
   GP2:
	UF : 1, UT : 1,
	J1=   -90.000 deg,	J2=   -90.000 deg
};
P[322]{
   GP1:
	UF : 1, UT : 1,		CONFIG : 'N U T, 0, 0, 0',
	X =  2873.686  mm,	Y =   257.161  mm,	Z =   290.593  mm,
	W =    15.416 deg,	P =   -27.050 deg,	R =   -31.230 deg
   GP2:
	UF : 1, UT : 1,
	J1=    90.000 deg,	J2=   135.000 deg
};
P[323]{
   GP1:
	UF : 1, UT : 1,		CONFIG : 'N U T, 0, 0, 0',
	X =  2382.956  mm,	Y =   364.175  mm,	Z =   194.044  mm,
	W =     1.770 deg,	P =     -.218 deg,	R =     7.120 deg
   GP2:
	UF : 1, UT : 1,
	J1=    90.000 deg,	J2=   135.000 deg
};
P[324]{
   GP1:
	UF : 1, UT : 1,		CONFIG : 'N U T, 0, 0, 0',
	X =  2754.103  mm,	Y =   362.637  mm,	Z =   193.804  mm,
	W =     1.712 deg,	P =    -2.514 deg,	R =     7.127 deg
   GP2:
	UF : 1, UT : 1,
	J1=    90.000 deg,	J2=   135.000 deg
};
P[325]{
   GP1:
	UF : 1, UT : 1,		CONFIG : 'N U T, 0, 0, 0',
	X =  1689.534  mm,	Y =    58.571  mm,	Z =   -13.480  mm,
	W =   -44.901 deg,	P =    -3.364 deg,	R =    -3.371 deg
   GP2:
	UF : 1, UT : 1,
	J1=    90.000 deg,	J2=    90.000 deg
};
P[326]{
   GP1:
	UF : 1, UT : 1,		CONFIG : 'N U T, 0, 0, 0',
	X =  1649.374  mm,	Y =    58.882  mm,	Z =   -13.998  mm,
	W =   -44.890 deg,	P =    -3.365 deg,	R =    -8.380 deg
   GP2:
	UF : 1, UT : 1,
	J1=    90.000 deg,	J2=    90.000 deg
};
P[327]{
   GP1:
	UF : 1, UT : 1,		CONFIG : 'N U T, 0, 0, 0',
	X =  1642.250  mm,	Y =    60.164  mm,	Z =   -14.447  mm,
	W =   -44.900 deg,	P =    -3.364 deg,	R =   -25.144 deg
   GP2:
	UF : 1, UT : 1,
	J1=    90.000 deg,	J2=    90.000 deg
};
P[328]{
   GP1:
	UF : 1, UT : 1,		CONFIG : 'N U T, 0, 0, 0',
	X =  1773.620  mm,	Y =   686.210  mm,	Z =   890.848  mm,
	W =     3.495 deg,	P =   -44.893 deg,	R =   -32.945 deg
   GP2:
	UF : 1, UT : 1,
	J1=   -90.000 deg,	J2=   -90.000 deg
};
P[329]{
   GP1:
	UF : 1, UT : 1,		CONFIG : 'N U T, 0, 0, 0',
	X =  1621.076  mm,	Y =   252.669  mm,	Z =   917.633  mm,
	W =    44.253 deg,	P =    -9.164 deg,	R =   -44.759 deg
   GP2:
	UF : 1, UT : 1,
	J1=   -90.000 deg,	J2=   -90.000 deg
};
P[330]{
   GP1:
	UF : 1, UT : 1,		CONFIG : 'N U T, 0, 0, 0',
	X =  1636.319  mm,	Y =    65.730  mm,	Z =   -14.946  mm,
	W =   -44.390 deg,	P =     8.298 deg,	R =   -38.036 deg
   GP2:
	UF : 1, UT : 1,
	J1=    90.000 deg,	J2=    90.000 deg
};
P[331]{
   GP1:
	UF : 1, UT : 1,		CONFIG : 'N U T, 0, 0, 0',
	X =  1604.762  mm,	Y =    95.897  mm,	Z =   -15.933  mm,
	W =   -44.391 deg,	P =     8.298 deg,	R =   -36.615 deg
   GP2:
	UF : 1, UT : 1,
	J1=    90.000 deg,	J2=    90.000 deg
};
P[332]{
   GP1:
	UF : 1, UT : 1,		CONFIG : 'N U T, 0, 0, 0',
	X =  1583.448  mm,	Y =   103.630  mm,	Z =   -15.279  mm,
	W =   -46.365 deg,	P =   -21.592 deg,	R =   -12.091 deg
   GP2:
	UF : 1, UT : 1,
	J1=    90.000 deg,	J2=    90.000 deg
};
P[333]{
   GP1:
	UF : 1, UT : 1,		CONFIG : 'N U T, 0, 0, 0',
	X =  1563.530  mm,	Y =    78.943  mm,	Z =   -13.367  mm,
	W =    32.003 deg,	P =   -33.504 deg,	R =   -53.547 deg
   GP2:
	UF : 1, UT : 1,
	J1=    90.000 deg,	J2=    90.000 deg
};
P[334]{
   GP1:
	UF : 1, UT : 1,		CONFIG : 'N U T, 0, 0, 0',
	X =  1761.847  mm,	Y =   175.594  mm,	Z =   881.529  mm,
	W =    53.651 deg,	P =   -10.142 deg,	R =   -83.497 deg
   GP2:
	UF : 1, UT : 1,
	J1=   -90.000 deg,	J2=   -90.000 deg
};
P[335]{
   GP1:
	UF : 1, UT : 1,		CONFIG : 'N U T, 0, 0, 0',
	X =  1298.520  mm,	Y =   205.285  mm,	Z =   914.227  mm,
	W =    53.651 deg,	P =   -10.142 deg,	R =   -83.497 deg
   GP2:
	UF : 1, UT : 1,
	J1=   -90.000 deg,	J2=   -90.000 deg
};
P[336]{
   GP1:
	UF : 1, UT : 1,		CONFIG : 'N U T, 0, 0, 0',
	X =  1138.188  mm,	Y =  -401.770  mm,	Z =  1054.451  mm,
	W =    41.557 deg,	P =   -19.100 deg,	R =   -69.755 deg
   GP2:
	UF : 1, UT : 1,
	J1=   -90.000 deg,	J2=    90.000 deg
};
P[337]{
   GP1:
	UF : 1, UT : 1,		CONFIG : 'N U T, 0, 0, 0',
	X =  1293.188  mm,	Y =  -401.770  mm,	Z =  1054.451  mm,
	W =    41.557 deg,	P =   -19.100 deg,	R =   -69.755 deg
   GP2:
	UF : 1, UT : 1,
	J1=   -90.000 deg,	J2=    90.000 deg
};
P[338]{
   GP1:
	UF : 1, UT : 1,		CONFIG : 'N U T, 0, 0, 0',
	X =  1645.188  mm,	Y =  -324.770  mm,	Z =   895.451  mm,
	W =    32.845 deg,	P =   -32.685 deg,	R =   -50.103 deg
   GP2:
	UF : 1, UT : 1,
	J1=   -90.000 deg,	J2=    90.000 deg
};
P[339]{
   GP1:
	UF : 1, UT : 1,		CONFIG : 'N U T, 0, 0, 0',
	X =  1558.407  mm,	Y =    32.303  mm,	Z =   -12.858  mm,
	W =    32.003 deg,	P =   -33.504 deg,	R =   -53.546 deg
   GP2:
	UF : 1, UT : 1,
	J1=    90.000 deg,	J2=    90.000 deg
};
P[340]{
   GP1:
	UF : 1, UT : 1,		CONFIG : 'N U T, 0, 0, 0',
	X =  1556.004  mm,	Y =    26.319  mm,	Z =   -12.970  mm,
	W =    32.004 deg,	P =   -33.504 deg,	R =   -81.670 deg
   GP2:
	UF : 1, UT : 1,
	J1=    90.000 deg,	J2=    90.000 deg
};
P[341]{
   GP1:
	UF : 1, UT : 1,		CONFIG : 'N U T, 0, 0, 0',
	X =  1548.265  mm,	Y =    23.382  mm,	Z =   -13.500  mm,
	W =    32.004 deg,	P =   -33.504 deg,	R =  -110.246 deg
   GP2:
	UF : 1, UT : 1,
	J1=    90.000 deg,	J2=    90.000 deg
};
P[342]{
   GP1:
	UF : 1, UT : 1,		CONFIG : 'N U T, 0, 0, 0',
	X =  1541.836  mm,	Y =    22.683  mm,	Z =   -13.499  mm,
	W =    32.004 deg,	P =   -33.504 deg,	R =  -110.246 deg
   GP2:
	UF : 1, UT : 1,
	J1=    90.000 deg,	J2=    90.000 deg
};
P[343]{
   GP1:
	UF : 1, UT : 1,		CONFIG : 'N U T, 0, 0, 0',
	X =  2750.935  mm,	Y =  -367.697  mm,	Z =   194.122  mm,
	W =    -4.046 deg,	P =     -.974 deg,	R =   -13.560 deg
   GP2:
	UF : 1, UT : 1,
	J1=    90.000 deg,	J2=  -135.000 deg
};
P[344]{
   GP1:
	UF : 1, UT : 1,		CONFIG : 'N U T, 0, 0, 0',
	X =  1707.928  mm,	Y =  -697.784  mm,	Z =   947.079  mm,
	W =    40.895 deg,	P =   -20.702 deg,	R =   -39.796 deg
   GP2:
	UF : 1, UT : 1,
	J1=   -90.000 deg,	J2=    90.000 deg
};
P[345]{
   GP1:
	UF : 1, UT : 1,		CONFIG : 'N U T, 0, 0, 0',
	X =  1651.323  mm,	Y =  -246.754  mm,	Z =   908.002  mm,
	W =   -48.803 deg,	P =   -10.122 deg,	R =    46.350 deg
   GP2:
	UF : 1, UT : 1,
	J1=   -90.000 deg,	J2=    90.000 deg
};
P[346]{
   GP1:
	UF : 1, UT : 1,		CONFIG : 'N U T, 0, 0, 0',
	X =  2067.448  mm,	Y =   -40.115  mm,	Z =    22.547  mm,
	W =    34.294 deg,	P =    -8.375 deg,	R =   -88.174 deg
   GP2:
	UF : 1, UT : 1,
	J1=    80.000 deg,	J2=   -90.000 deg
};
P[347]{
   GP1:
	UF : 1, UT : 1,		CONFIG : 'N U T, 0, 0, 0',
	X =  2071.895  mm,	Y =    -9.046  mm,	Z =    21.479  mm,
	W =    34.239 deg,	P =    -8.411 deg,	R =   -88.218 deg
   GP2:
	UF : 1, UT : 1,
	J1=    80.000 deg,	J2=   -90.000 deg
};
P[348]{
   GP1:
	UF : 1, UT : 1,		CONFIG : 'N U T, 0, 0, 0',
	X =  2076.271  mm,	Y =     4.342  mm,	Z =    21.635  mm,
	W =    30.086 deg,	P =   -21.642 deg,	R =   -96.023 deg
   GP2:
	UF : 1, UT : 1,
	J1=    80.000 deg,	J2=   -90.000 deg
};
P[349]{
   GP1:
	UF : 1, UT : 1,		CONFIG : 'N U T, 0, 0, 0',
	X =  2086.260  mm,	Y =    16.914  mm,	Z =    21.636  mm,
	W =    23.411 deg,	P =   -33.701 deg,	R =  -102.541 deg
   GP2:
	UF : 1, UT : 1,
	J1=    80.000 deg,	J2=   -90.000 deg
};
P[350]{
   GP1:
	UF : 1, UT : 1,		CONFIG : 'N U T, 0, 0, 0',
	X =  1747.472  mm,	Y =  -189.520  mm,	Z =   887.139  mm,
	W =   -45.012 deg,	P =   -17.288 deg,	R =    71.040 deg
   GP2:
	UF : 1, UT : 1,
	J1=   -90.000 deg,	J2=    90.000 deg
};
P[351]{
   GP1:
	UF : 1, UT : 1,		CONFIG : 'N U T, 0, 0, 0',
	X =  1268.443  mm,	Y =  -269.816  mm,	Z =   903.959  mm,
	W =   -45.005 deg,	P =   -17.287 deg,	R =    72.332 deg
   GP2:
	UF : 1, UT : 1,
	J1=   -90.000 deg,	J2=    90.000 deg
};
P[352]{
   GP1:
	UF : 1, UT : 1,		CONFIG : 'N U B, 0, 0, 0',
	X =   357.030  mm,	Y =     -.134  mm,	Z =  2422.493  mm,
	W =     -.020 deg,	P =   -39.773 deg,	R =      .020 deg
   GP2:
	UF : 1, UT : 1,
	J1=    90.000 deg,	J2=    90.000 deg
};
P[353]{
   GP1:
	UF : 1, UT : 1,		CONFIG : 'N U T, 0, 0, 0',
	X =  1748.616  mm,	Y =   271.230  mm,	Z =  1366.022  mm,
	W =     -.010 deg,	P =    45.000 deg,	R =    57.110 deg
   GP2:
	UF : 1, UT : 1,
	J1=    90.000 deg,	J2=    90.000 deg
};
P[354]{
   GP1:
	UF : 1, UT : 1,		CONFIG : 'N U T, 0, 0, 0',
	X =  2361.616  mm,	Y =    71.231  mm,	Z =   946.022  mm,
	W =   -25.245 deg,	P =    38.577 deg,	R =    56.316 deg
   GP2:
	UF : 1, UT : 1,
	J1=    90.000 deg,	J2=    90.000 deg
};
P[355]{
   GP1:
	UF : 1, UT : 1,		CONFIG : 'N U T, 0, 0, 0',
	X =  2099.624  mm,	Y =    22.343  mm,	Z =    16.408  mm,
	W =    23.412 deg,	P =   -33.704 deg,	R =  -102.541 deg
   GP2:
	UF : 1, UT : 1,
	J1=    80.000 deg,	J2=   -90.000 deg
};
P[356]{
   GP1:
	UF : 1, UT : 1,		CONFIG : 'N U T, 0, 0, -1',
	X =  1652.850  mm,	Y =  -150.757  mm,	Z =   -11.674  mm,
	W =   -35.869 deg,	P =    29.235 deg,	R =   125.842 deg
   GP2:
	UF : 1, UT : 1,
	J1=    90.000 deg,	J2=    90.000 deg
};
P[357]{
   GP1:
	UF : 1, UT : 1,		CONFIG : 'N U T, 0, 0, 0',
	X =  2422.384  mm,	Y =    34.711  mm,	Z =   895.214  mm,
	W =   -26.680 deg,	P =    37.686 deg,	R =    50.517 deg
   GP2:
	UF : 1, UT : 1,
	J1=    90.000 deg,	J2=    90.000 deg
};
P[358]{
   GP1:
	UF : 1, UT : 1,		CONFIG : 'N U T, 0, 0, 0',
	X =  2455.577  mm,	Y =   -29.126  mm,	Z =   895.215  mm,
	W =   -37.503 deg,	P =    26.957 deg,	R =   -56.583 deg
   GP2:
	UF : 1, UT : 1,
	J1=    90.000 deg,	J2=    90.000 deg
};
P[359]{
   GP1:
	UF : 1, UT : 1,		CONFIG : 'N U T, 0, 0, 0',
	X =  1656.099  mm,	Y =    18.125  mm,	Z =   -14.737  mm,
	W =   -35.780 deg,	P =    29.286 deg,	R =   139.578 deg
   GP2:
	UF : 1, UT : 1,
	J1=    89.999 deg,	J2=    90.000 deg
};
P[360]{
   GP1:
	UF : 1, UT : 1,		CONFIG : 'N U T, 0, 0, 0',
	X =  2354.497  mm,	Y =   -22.564  mm,	Z =     1.025  mm,
	W =    44.702 deg,	P =     5.823 deg,	R =    -5.853 deg
   GP2:
	UF : 1, UT : 1,
	J1=    90.000 deg,	J2=    90.000 deg
};
P[361]{
   GP1:
	UF : 1, UT : 1,		CONFIG : 'N U T, 0, 0, 0',
	X =  2456.027  mm,	Y =   -61.584  mm,	Z =   962.417  mm,
	W =   -36.666 deg,	P =    28.172 deg,	R =   -57.618 deg
   GP2:
	UF : 1, UT : 1,
	J1=    90.000 deg,	J2=    90.000 deg
};
P[362]{
   GP1:
	UF : 1, UT : 1,		CONFIG : 'N U T, 0, 0, 0',
	X =  2083.492  mm,	Y =   163.430  mm,	Z =  1073.319  mm,
	W =   -10.584 deg,	P =    13.460 deg,	R =   -52.492 deg
   GP2:
	UF : 1, UT : 1,
	J1=    90.000 deg,	J2=    90.000 deg
};
P[363]{
   GP1:
	UF : 1, UT : 1,		CONFIG : 'N U T, 0, 0, 0',
	X =  2865.354  mm,	Y =  1371.120  mm,	Z =    76.936  mm,
	W =    -1.528 deg,	P =    -1.642 deg,	R =     2.928 deg
   GP2:
	UF : 1, UT : 1,
	J1=    94.999 deg,	J2=    90.000 deg
};
P[364]{
   GP1:
	UF : 1, UT : 1,		CONFIG : 'N U T, 0, 0, 0',
	X =  1411.479  mm,	Y =   569.332  mm,	Z =  1273.375  mm,
	W =    35.032 deg,	P =    -9.420 deg,	R =   -62.796 deg
   GP2:
	UF : 1, UT : 1,
	J1=    90.000 deg,	J2=    90.000 deg
};
P[365]{
   GP1:
	UF : 1, UT : 1,		CONFIG : 'N U T, 0, 0, 0',
	X =  1411.479  mm,	Y =   569.333  mm,	Z =   491.080  mm,
	W =   -35.557 deg,	P =    -4.844 deg,	R =      .283 deg
   GP2:
	UF : 1, UT : 1,
	J1=    90.000 deg,	J2=   100.000 deg
};
P[366]{
   GP1:
	UF : 1, UT : 1,		CONFIG : 'N U T, 0, 0, 0',
	X =  2503.479  mm,	Y =   301.762  mm,	Z =   250.437  mm,
	W =   -27.790 deg,	P =   -29.118 deg,	R =   -29.928 deg
   GP2:
	UF : 1, UT : 1,
	J1=    90.000 deg,	J2=   100.000 deg
};
P[367]{
   GP1:
	UF : 1, UT : 1,		CONFIG : 'N U T, 0, 0, 0',
	X =  2523.555  mm,	Y =   176.173  mm,	Z =   166.469  mm,
	W =   -19.929 deg,	P =   -29.386 deg,	R =   -53.539 deg
   GP2:
	UF : 1, UT : 1,
	J1=    90.000 deg,	J2=   100.000 deg
};
P[368]{
   GP1:
	UF : 1, UT : 1,		CONFIG : 'N U T, 0, 0, 0',
	X =  2525.579  mm,	Y =   -21.476  mm,	Z =     3.467  mm,
	W =    44.791 deg,	P =    -4.849 deg,	R =     4.871 deg
   GP2:
	UF : 1, UT : 1,
	J1=    90.000 deg,	J2=    90.000 deg
};
P[369]{
   GP1:
	UF : 1, UT : 1,		CONFIG : 'N U T, 0, 0, 0',
	X =  2355.026  mm,	Y =    67.774  mm,	Z =     -.631  mm,
	W =    44.702 deg,	P =     5.823 deg,	R =    -9.844 deg
   GP2:
	UF : 1, UT : 1,
	J1=    90.000 deg,	J2=    90.000 deg
};
P[370]{
   GP1:
	UF : 1, UT : 1,		CONFIG : 'N U T, 0, 0, 0',
	X =  2401.530  mm,	Y =    69.488  mm,	Z =    -1.003  mm,
	W =    44.700 deg,	P =     5.824 deg,	R =    -9.846 deg
   GP2:
	UF : 1, UT : 1,
	J1=    90.000 deg,	J2=    90.000 deg
};
P[371]{
   GP1:
	UF : 1, UT : 1,		CONFIG : 'N U T, 0, 0, 0',
	X =  2504.982  mm,	Y =    92.808  mm,	Z =    48.278  mm,
	W =   -29.361 deg,	P =   -19.966 deg,	R =   -47.133 deg
   GP2:
	UF : 1, UT : 1,
	J1=    90.000 deg,	J2=   100.000 deg
};
P[372]{
   GP1:
	UF : 1, UT : 1,		CONFIG : 'N U T, 0, 0, 0',
	X =  2503.480  mm,	Y =   301.761  mm,	Z =   230.080  mm,
	W =   -25.716 deg,	P =   -28.362 deg,	R =   -30.253 deg
   GP2:
	UF : 1, UT : 1,
	J1=    90.000 deg,	J2=   100.000 deg
};
P[373]{
   GP1:
	UF : 1, UT : 1,		CONFIG : 'N U T, 0, 0, 0',
	X =  2353.479  mm,	Y =   301.761  mm,	Z =   230.080  mm,
	W =   -28.643 deg,	P =   -22.532 deg,	R =   -28.032 deg
   GP2:
	UF : 1, UT : 1,
	J1=    90.000 deg,	J2=   100.000 deg
};
P[374]{
   GP1:
	UF : 1, UT : 1,		CONFIG : 'N U T, 0, 0, 0',
	X =  2353.479  mm,	Y =   121.761  mm,	Z =    98.080  mm,
	W =   -35.259 deg,	P =    -6.903 deg,	R =    -2.628 deg
   GP2:
	UF : 1, UT : 1,
	J1=    90.000 deg,	J2=   100.000 deg
};
P[375]{
   GP1:
	UF : 1, UT : 1,		CONFIG : 'N U T, 0, 0, 0',
	X =  2426.517  mm,	Y =    66.846  mm,	Z =     2.875  mm,
	W =    43.736 deg,	P =   -11.847 deg,	R =   -16.338 deg
   GP2:
	UF : 1, UT : 1,
	J1=    90.000 deg,	J2=    90.000 deg
};
P[376]{
   GP1:
	UF : 1, UT : 1,		CONFIG : 'N U T, 0, 0, 0',
	X =  2835.246  mm,	Y =  1480.319  mm,	Z =   893.361  mm,
	W =     1.884 deg,	P =   -42.060 deg,	R =    -2.906 deg
   GP2:
	UF : 1, UT : 1,
	J1=    95.000 deg,	J2=    90.000 deg
};
P[377]{
   GP1:
	UF : 1, UT : 1,		CONFIG : 'N U T, 0, 0, 0',
	X =  2354.014  mm,	Y =   141.761  mm,	Z =   162.390  mm,
	W =   -30.293 deg,	P =   -21.076 deg,	R =     2.382 deg
   GP2:
	UF : 1, UT : 1,
	J1=    90.000 deg,	J2=   100.000 deg
};
P[378]{
   GP1:
	UF : 1, UT : 1,		CONFIG : 'N U T, 0, 0, 0',
	X =  1657.674  mm,	Y =   274.797  mm,	Z =   284.639  mm,
	W =   -30.355 deg,	P =    -3.481 deg,	R =     2.192 deg
   GP2:
	UF : 1, UT : 1,
	J1=    90.000 deg,	J2=   100.000 deg
};
P[379]{
   GP1:
	UF : 1, UT : 1,		CONFIG : 'N U T, 0, 0, 0',
	X =  1192.015  mm,	Y =   363.761  mm,	Z =  1100.390  mm,
	W =     1.467 deg,	P =    42.180 deg,	R =    96.897 deg
   GP2:
	UF : 1, UT : 1,
	J1=    90.000 deg,	J2=    90.000 deg
};
P[380]{
   GP1:
	UF : 1, UT : 1,		CONFIG : 'N U T, 0, 0, 0',
	X =  2149.186  mm,	Y =   260.397  mm,	Z =  1100.389  mm,
	W =    -5.363 deg,	P =    30.946 deg,	R =    85.742 deg
   GP2:
	UF : 1, UT : 1,
	J1=    90.000 deg,	J2=    90.000 deg
};
P[381]{
   GP1:
	UF : 1, UT : 1,		CONFIG : 'N U T, 0, 0, 0',
	X =  2149.186  mm,	Y =   260.397  mm,	Z =   900.389  mm,
	W =    -6.655 deg,	P =    43.605 deg,	R =    84.955 deg
   GP2:
	UF : 1, UT : 1,
	J1=    90.000 deg,	J2=    90.000 deg
};
P[382]{
   GP1:
	UF : 1, UT : 1,		CONFIG : 'N U T, 0, 0, 0',
	X =  2834.470  mm,	Y =  1506.572  mm,	Z =   893.930  mm,
	W =      .428 deg,	P =   -42.104 deg,	R =     -.755 deg
   GP2:
	UF : 1, UT : 1,
	J1=    95.000 deg,	J2=    90.000 deg
};
P[383]{
   GP1:
	UF : 1, UT : 1,		CONFIG : 'N U T, 0, 0, 0',
	X =  2826.478  mm,	Y =  1533.650  mm,	Z =   892.309  mm,
	W =    47.771 deg,	P =   -12.839 deg,	R =   -44.177 deg
   GP2:
	UF : 1, UT : 1,
	J1=    95.000 deg,	J2=    90.000 deg
};
P[384]{
   GP1:
	UF : 1, UT : 1,		CONFIG : 'N U T, 0, 0, 0',
	X =  2815.159  mm,	Y =  1553.063  mm,	Z =   888.714  mm,
	W =    47.469 deg,	P =    -2.511 deg,	R =   -28.096 deg
   GP2:
	UF : 1, UT : 1,
	J1=    95.000 deg,	J2=    90.000 deg
};
P[385]{
   GP1:
	UF : 1, UT : 1,		CONFIG : 'N U T, 0, 0, 0',
	X =  2769.546  mm,	Y =  1573.155  mm,	Z =   887.864  mm,
	W =    47.469 deg,	P =    -2.511 deg,	R =   -28.096 deg
   GP2:
	UF : 1, UT : 1,
	J1=    95.000 deg,	J2=    90.000 deg
};
P[386]{
   GP1:
	UF : 1, UT : 1,		CONFIG : 'N U T, 0, 0, 0',
	X =  2763.445  mm,	Y =  1576.537  mm,	Z =   885.675  mm,
	W =    46.964 deg,	P =     8.280 deg,	R =   -26.942 deg
   GP2:
	UF : 1, UT : 1,
	J1=    95.000 deg,	J2=    90.000 deg
};
P[387]{
   GP1:
	UF : 1, UT : 1,		CONFIG : 'N U T, 0, 0, 0',
	X =  2755.656  mm,	Y =  1578.479  mm,	Z =   883.891  mm,
	W =    46.312 deg,	P =    12.118 deg,	R =   -20.583 deg
   GP2:
	UF : 1, UT : 1,
	J1=    95.000 deg,	J2=    90.000 deg
};
P[388]{
   GP1:
	UF : 1, UT : 1,		CONFIG : 'N U T, 0, 0, 0',
	X =  2718.475  mm,	Y =  1577.296  mm,	Z =   882.326  mm,
	W =    46.312 deg,	P =    12.119 deg,	R =   -20.583 deg
   GP2:
	UF : 1, UT : 1,
	J1=    95.000 deg,	J2=    90.000 deg
};
P[389]{
   GP1:
	UF : 1, UT : 1,		CONFIG : 'N U T, 0, 0, 0',
	X =  1681.503  mm,	Y =   305.740  mm,	Z =   839.267  mm,
	W =     3.505 deg,	P =   -44.886 deg,	R =    -9.395 deg
   GP2:
	UF : 1, UT : 1,
	J1=   -90.000 deg,	J2=   -90.000 deg
};
P[390]{
   GP1:
	UF : 1, UT : 1,		CONFIG : 'N U T, 0, 0, 0',
	X =  2629.170  mm,	Y =    65.409  mm,	Z =   972.111  mm,
	W =   -34.833 deg,	P =    25.325 deg,	R =    61.817 deg
   GP2:
	UF : 1, UT : 1,
	J1=    90.000 deg,	J2=    90.000 deg
};
P[391]{
   GP1:
	UF : 1, UT : 1,		CONFIG : 'N U T, 0, 0, 0',
	X =  2125.926  mm,	Y =   140.894  mm,	Z =   972.130  mm,
	W =      .934 deg,	P =    44.201 deg,	R =   163.009 deg
   GP2:
	UF : 1, UT : 1,
	J1=    90.000 deg,	J2=    90.000 deg
};
P[392]{
   GP1:
	UF : 1, UT : 1,		CONFIG : 'N U T, 0, 0, 0',
	X =  1682.513  mm,	Y =   318.688  mm,	Z =   839.335  mm,
	W =     3.495 deg,	P =   -44.892 deg,	R =    -9.388 deg
   GP2:
	UF : 1, UT : 1,
	J1=   -90.000 deg,	J2=   -90.000 deg
};
P[393]{
   GP1:
	UF : 1, UT : 1,		CONFIG : 'N U T, 0, 0, 0',
	X =  1683.114  mm,	Y =   324.974  mm,	Z =   839.334  mm,
	W =     3.495 deg,	P =   -44.893 deg,	R =   -17.009 deg
   GP2:
	UF : 1, UT : 1,
	J1=   -90.000 deg,	J2=   -90.000 deg
};
P[394]{
   GP1:
	UF : 1, UT : 1,		CONFIG : 'N U T, 0, 0, 0',
	X =  1684.099  mm,	Y =   331.260  mm,	Z =   839.334  mm,
	W =     3.495 deg,	P =   -44.893 deg,	R =   -22.694 deg
   GP2:
	UF : 1, UT : 1,
	J1=   -90.000 deg,	J2=   -90.000 deg
};
P[395]{
   GP1:
	UF : 1, UT : 1,		CONFIG : 'N U T, 0, 0, 0',
	X =  1707.379  mm,	Y =   402.340  mm,	Z =   838.425  mm,
	W =     3.495 deg,	P =   -44.893 deg,	R =   -22.694 deg
   GP2:
	UF : 1, UT : 1,
	J1=   -90.000 deg,	J2=   -90.000 deg
};
P[396]{
   GP1:
	UF : 1, UT : 1,		CONFIG : 'N U T, 0, 0, 0',
	X =  1708.479  mm,	Y =   405.840  mm,	Z =   838.426  mm,
	W =     3.495 deg,	P =   -44.893 deg,	R =   -29.180 deg
   GP2:
	UF : 1, UT : 1,
	J1=   -90.000 deg,	J2=   -90.000 deg
};
P[397]{
   GP1:
	UF : 1, UT : 1,		CONFIG : 'N U T, 0, 0, 0',
	X =  1710.366  mm,	Y =   410.197  mm,	Z =   838.426  mm,
	W =     3.495 deg,	P =   -44.893 deg,	R =   -32.945 deg
   GP2:
	UF : 1, UT : 1,
	J1=   -90.000 deg,	J2=   -90.000 deg
};
P[398]{
   GP1:
	UF : 1, UT : 1,		CONFIG : 'N U T, 0, 0, 0',
	X =  1848.308  mm,	Y =   668.682  mm,	Z =   838.425  mm,
	W =     3.495 deg,	P =   -44.893 deg,	R =   -32.945 deg
   GP2:
	UF : 1, UT : 1,
	J1=   -90.000 deg,	J2=   -90.000 deg
};
P[399]{
   GP1:
	UF : 1, UT : 1,		CONFIG : 'N U T, 0, 0, 0',
	X =  1912.100  mm,	Y =   218.688  mm,	Z =  1134.610  mm,
	W =    29.171 deg,	P =    60.290 deg,	R =  -156.347 deg
   GP2:
	UF : 1, UT : 1,
	J1=    90.000 deg,	J2=    90.000 deg
};
P[400]{
   GP1:
	UF : 1, UT : 1,		CONFIG : 'N U T, 0, 0, 1',
	X =   967.194  mm,	Y =   236.168  mm,	Z =  1196.476  mm,
	W =   -52.081 deg,	P =    56.220 deg,	R =   149.523 deg
   GP2:
	UF : 1, UT : 1,
	J1=    80.000 deg,	J2=    90.000 deg
};
P[401]{
   GP1:
	UF : 1, UT : 1,		CONFIG : 'N U T, 0, 0, 0',
	X =  1113.896  mm,	Y =  -312.111  mm,	Z =   774.061  mm,
	W =   -55.009 deg,	P =    11.243 deg,	R =   103.085 deg
   GP2:
	UF : 1, UT : 1,
	J1=    80.000 deg,	J2=    90.000 deg
};
P[402]{
   GP1:
	UF : 1, UT : 1,		CONFIG : 'N U T, 0, 0, 0',
	X =  2001.132  mm,	Y =  -144.328  mm,	Z =   162.948  mm,
	W =   -38.656 deg,	P =   -14.170 deg,	R =   113.061 deg
   GP2:
	UF : 1, UT : 1,
	J1=    80.000 deg,	J2=    90.000 deg
};
P[403]{
   GP1:
	UF : 1, UT : 1,		CONFIG : 'N U T, 0, 0, 0',
	X =  1716.035  mm,	Y =   257.698  mm,	Z =   837.982  mm,
	W =    44.762 deg,	P =    -3.344 deg,	R =   -39.059 deg
   GP2:
	UF : 1, UT : 1,
	J1=   -90.000 deg,	J2=   -90.000 deg
};
P[404]{
   GP1:
	UF : 1, UT : 1,		CONFIG : 'N U T, 0, 0, 0',
	X =  1821.570  mm,	Y =   170.709  mm,	Z =   839.692  mm,
	W =    43.945 deg,	P =    -9.912 deg,	R =   -48.939 deg
   GP2:
	UF : 1, UT : 1,
	J1=   -90.000 deg,	J2=   -90.000 deg
};
P[405]{
   GP1:
	UF : 1, UT : 1,		CONFIG : 'N U T, 0, 0, 0',
	X =  1848.071  mm,	Y =   149.119  mm,	Z =   839.997  mm,
	W =    42.189 deg,	P =   -16.814 deg,	R =   -52.365 deg
   GP2:
	UF : 1, UT : 1,
	J1=   -90.000 deg,	J2=   -90.000 deg
};
P[406]{
   GP1:
	UF : 1, UT : 1,		CONFIG : 'N U T, 0, 0, 0',
	X =  1866.284  mm,	Y =   133.819  mm,	Z =   839.998  mm,
	W =    42.189 deg,	P =   -16.814 deg,	R =   -63.440 deg
   GP2:
	UF : 1, UT : 1,
	J1=   -90.000 deg,	J2=   -90.000 deg
};
P[407]{
   GP1:
	UF : 1, UT : 1,		CONFIG : 'N U T, 0, 0, 0',
	X =  1679.887  mm,	Y =  -309.053  mm,	Z =   840.871  mm,
	W =    32.859 deg,	P =   -32.671 deg,	R =   -50.113 deg
   GP2:
	UF : 1, UT : 1,
	J1=   -90.000 deg,	J2=    90.000 deg
};
P[408]{
   GP1:
	UF : 1, UT : 1,		CONFIG : 'N U T, 0, 0, 0',
	X =  1681.832  mm,	Y =  -318.985  mm,	Z =   840.951  mm,
	W =    32.845 deg,	P =   -32.685 deg,	R =   -50.103 deg
   GP2:
	UF : 1, UT : 1,
	J1=   -90.000 deg,	J2=    90.000 deg
};
P[409]{
   GP1:
	UF : 1, UT : 1,		CONFIG : 'N U T, 0, 0, 0',
	X =  1681.832  mm,	Y =  -323.128  mm,	Z =   840.950  mm,
	W =    32.845 deg,	P =   -32.685 deg,	R =   -45.680 deg
   GP2:
	UF : 1, UT : 1,
	J1=   -90.000 deg,	J2=    90.000 deg
};
P[410]{
   GP1:
	UF : 1, UT : 1,		CONFIG : 'N U T, 0, 0, 0',
	X =  1682.484  mm,	Y =  -329.978  mm,	Z =   840.955  mm,
	W =    32.851 deg,	P =   -32.684 deg,	R =   -43.121 deg
   GP2:
	UF : 1, UT : 1,
	J1=   -90.000 deg,	J2=    90.000 deg
};
P[411]{
   GP1:
	UF : 1, UT : 1,		CONFIG : 'N U T, 0, 0, 0',
	X =  1707.241  mm,	Y =  -405.978  mm,	Z =   840.954  mm,
	W =    32.851 deg,	P =   -32.684 deg,	R =   -43.121 deg
   GP2:
	UF : 1, UT : 1,
	J1=   -90.000 deg,	J2=    90.000 deg
};
P[412]{
   GP1:
	UF : 1, UT : 1,		CONFIG : 'N U T, 0, 0, 0',
	X =  1708.270  mm,	Y =  -409.406  mm,	Z =   840.955  mm,
	W =    32.851 deg,	P =   -32.684 deg,	R =   -40.021 deg
   GP2:
	UF : 1, UT : 1,
	J1=   -90.000 deg,	J2=    90.000 deg
};
P[413]{
   GP1:
	UF : 1, UT : 1,		CONFIG : 'N U T, 0, 0, 0',
	X =  2574.769  mm,	Y =  -572.619  mm,	Z =   -35.483  mm,
	W =   -30.992 deg,	P =   -17.135 deg,	R =    63.872 deg
   GP2:
	UF : 1, UT : 1,
	J1=    80.000 deg,	J2=    90.000 deg
};
P[414]{
   GP1:
	UF : 1, UT : 1,		CONFIG : 'N U T, 0, 0, 0',
	X =  2505.964  mm,	Y =  -686.865  mm,	Z =    -4.700  mm,
	W =   -27.895 deg,	P =   -22.051 deg,	R =    54.654 deg
   GP2:
	UF : 1, UT : 1,
	J1=    80.000 deg,	J2=    90.000 deg
};
P[415]{
   GP1:
	UF : 1, UT : 1,		CONFIG : 'N U T, 0, 0, 0',
	X =  1708.764  mm,	Y =  -412.653  mm,	Z =   840.603  mm,
	W =    37.851 deg,	P =   -26.432 deg,	R =   -42.977 deg
   GP2:
	UF : 1, UT : 1,
	J1=   -90.000 deg,	J2=    90.000 deg
};
P[416]{
   GP1:
	UF : 1, UT : 1,		CONFIG : 'N U T, 0, 0, 0',
	X =  1847.936  mm,	Y =  -669.624  mm,	Z =   840.603  mm,
	W =    37.851 deg,	P =   -26.432 deg,	R =   -42.976 deg
   GP2:
	UF : 1, UT : 1,
	J1=   -90.000 deg,	J2=    90.000 deg
};
P[417]{
   GP1:
	UF : 1, UT : 1,		CONFIG : 'N U T, 0, 0, 0',
	X =  1717.056  mm,	Y =  -256.503  mm,	Z =   837.218  mm,
	W =   -39.799 deg,	P =    -6.282 deg,	R =    41.707 deg
   GP2:
	UF : 1, UT : 1,
	J1=   -90.000 deg,	J2=    90.000 deg
};
P[418]{
   GP1:
	UF : 1, UT : 1,		CONFIG : 'N U T, 0, 0, 0',
	X =  1805.891  mm,	Y =  -184.307  mm,	Z =   837.201  mm,
	W =   -40.187 deg,	P =    -1.576 deg,	R =    52.566 deg
   GP2:
	UF : 1, UT : 1,
	J1=   -90.000 deg,	J2=    90.000 deg
};
P[419]{
   GP1:
	UF : 1, UT : 1,		CONFIG : 'N U T, 0, 0, 0',
	X =  1840.820  mm,	Y =  -155.377  mm,	Z =   837.200  mm,
	W =   -40.187 deg,	P =    -1.576 deg,	R =    63.074 deg
   GP2:
	UF : 1, UT : 1,
	J1=   -90.000 deg,	J2=    90.000 deg
};
P[420]{
   GP1:
	UF : 1, UT : 1,		CONFIG : 'N U T, 0, 0, 0',
	X =  1865.820  mm,	Y =  -134.434  mm,	Z =   837.199  mm,
	W =   -40.187 deg,	P =    -1.576 deg,	R =    78.005 deg
   GP2:
	UF : 1, UT : 1,
	J1=   -90.000 deg,	J2=    90.000 deg
};
P[421]{
   GP1:
	UF : 1, UT : 1,		CONFIG : 'N U T, 0, 0, 0',
	X =  2482.381  mm,	Y =  -565.789  mm,	Z =   129.772  mm,
	W =   -49.202 deg,	P =    -2.428 deg,	R =    64.376 deg
   GP2:
	UF : 1, UT : 1,
	J1=    80.000 deg,	J2=    90.000 deg
};
P[422]{
   GP1:
	UF : 1, UT : 1,		CONFIG : 'N U T, 0, 0, 0',
	X =  1315.952  mm,	Y =  -565.788  mm,	Z =   468.198  mm,
	W =   -49.202 deg,	P =    -2.428 deg,	R =    64.376 deg
   GP2:
	UF : 1, UT : 1,
	J1=    80.000 deg,	J2=    90.000 deg
};
P[423]{
   GP1:
	UF : 1, UT : 1,		CONFIG : 'N U T, 0, 0, 0',
	X =  1291.369  mm,	Y = -1688.719  mm,	Z =  1275.725  mm,
	W =   -48.540 deg,	P =   -14.944 deg,	R =    31.683 deg
   GP2:
	UF : 1, UT : 1,
	J1=   180.000 deg,	J2=  -125.000 deg
};
P[424]{
   GP1:
	UF : 1, UT : 1,		CONFIG : 'N U T, 0, 0, 0',
	X =  1516.478  mm,	Y =  -924.777  mm,	Z =   251.093  mm,
	W =   -43.355 deg,	P =    13.455 deg,	R =    91.500 deg
   GP2:
	UF : 1, UT : 1,
	J1=    90.000 deg,	J2=   -90.000 deg
};
P[425]{
   GP1:
	UF : 1, UT : 1,		CONFIG : 'N U T, 0, 0, 0',
	X =  1689.800  mm,	Y =  1215.643  mm,	Z =  1225.099  mm,
	W =    19.059 deg,	P =    -5.228 deg,	R =    -7.084 deg
   GP2:
	UF : 1, UT : 1,
	J1=    94.999 deg,	J2=    90.000 deg
};
P[426]{
   GP1:
	UF : 1, UT : 1,		CONFIG : 'N U T, 0, 0, 0',
	X =  2379.239  mm,	Y =  -951.992  mm,	Z =   112.055  mm,
	W =   -43.355 deg,	P =    13.455 deg,	R =   104.588 deg
   GP2:
	UF : 1, UT : 1,
	J1=    90.000 deg,	J2=   -90.000 deg
};
P[427]{
   GP1:
	UF : 1, UT : 1,		CONFIG : 'N U T, 0, 0, 0',
	X =  2332.553  mm,	Y =   -45.582  mm,	Z =   845.925  mm,
	W =   -24.408 deg,	P =    42.022 deg,	R =    55.121 deg
   GP2:
	UF : 1, UT : 1,
	J1=    90.000 deg,	J2=    90.000 deg
};
P[428]{
   GP1:
	UF : 1, UT : 1,		CONFIG : 'N U T, 0, 0, 0',
	X =  2408.424  mm,	Y =   -44.749  mm,	Z =   846.748  mm,
	W =   -24.460 deg,	P =    42.071 deg,	R =    55.079 deg
   GP2:
	UF : 1, UT : 1,
	J1=    90.000 deg,	J2=    90.000 deg
};
P[429]{
   GP1:
	UF : 1, UT : 1,		CONFIG : 'N U T, 0, 0, 1',
	X =  2149.602  mm,	Y = -1008.832  mm,	Z =   291.902  mm,
	W =   -43.358 deg,	P =    13.457 deg,	R =   121.686 deg
   GP2:
	UF : 1, UT : 1,
	J1=    90.000 deg,	J2=   -90.000 deg
};
P[430]{
   GP1:
	UF : 1, UT : 1,		CONFIG : 'N U T, 0, 0, 0',
	X =  1603.602  mm,	Y =  -724.496  mm,	Z =   291.902  mm,
	W =   -24.164 deg,	P =   -39.192 deg,	R =   -55.648 deg
   GP2:
	UF : 1, UT : 1,
	J1=    90.000 deg,	J2=   -90.000 deg
};
P[431]{
   GP1:
	UF : 1, UT : 1,		CONFIG : 'N U T, 0, 0, 0',
	X =  2431.602  mm,	Y =  -724.497  mm,	Z =   291.902  mm,
	W =   -19.487 deg,	P =   -41.401 deg,	R =   -37.471 deg
   GP2:
	UF : 1, UT : 1,
	J1=    90.000 deg,	J2=   -90.000 deg
};
P[432]{
   GP1:
	UF : 1, UT : 1,		CONFIG : 'N U T, 0, 0, 0',
	X =  2488.601  mm,	Y =  -724.497  mm,	Z =    58.902  mm,
	W =   -19.487 deg,	P =   -41.401 deg,	R =   -47.828 deg
   GP2:
	UF : 1, UT : 1,
	J1=    90.000 deg,	J2=   -90.000 deg
};
P[433]{
   GP1:
	UF : 1, UT : 1,		CONFIG : 'N U T, 0, 0, 0',
	X =  2406.463  mm,	Y =   -45.092  mm,	Z =   844.000  mm,
	W =   -36.666 deg,	P =    28.172 deg,	R =   -57.618 deg
   GP2:
	UF : 1, UT : 1,
	J1=    90.000 deg,	J2=    90.000 deg
};
P[434]{
   GP1:
	UF : 1, UT : 1,		CONFIG : 'N U T, 0, 0, 0',
	X =  2406.465  mm,	Y =   -74.992  mm,	Z =   843.998  mm,
	W =   -36.666 deg,	P =    28.172 deg,	R =   -57.618 deg
   GP2:
	UF : 1, UT : 1,
	J1=    90.000 deg,	J2=    90.000 deg
};
P[435]{
   GP1:
	UF : 1, UT : 1,		CONFIG : 'N U T, 0, 0, 0',
	X =  2488.601  mm,	Y =  -724.497  mm,	Z =    58.902  mm,
	W =   -19.487 deg,	P =   -41.401 deg,	R =   -47.828 deg
   GP2:
	UF : 1, UT : 1,
	J1=    90.000 deg,	J2=   -90.000 deg
};
P[436]{
   GP1:
	UF : 1, UT : 1,		CONFIG : 'N U T, 0, 0, 0',
	X =  2431.602  mm,	Y =  -724.497  mm,	Z =   291.902  mm,
	W =   -19.487 deg,	P =   -41.401 deg,	R =   -37.471 deg
   GP2:
	UF : 1, UT : 1,
	J1=    90.000 deg,	J2=   -90.000 deg
};
P[437]{
   GP1:
	UF : 1, UT : 1,		CONFIG : 'N U T, 0, 0, 0',
	X =  1603.602  mm,	Y =  -724.496  mm,	Z =   291.902  mm,
	W =   -24.164 deg,	P =   -39.192 deg,	R =   -55.648 deg
   GP2:
	UF : 1, UT : 1,
	J1=    90.000 deg,	J2=   -90.000 deg
};
P[438]{
   GP1:
	UF : 1, UT : 1,		CONFIG : 'N U T, 0, 0, 0',
	X =  1523.303  mm,	Y =  -411.413  mm,	Z =   309.664  mm,
	W =    30.908 deg,	P =   -20.021 deg,	R =    92.765 deg
   GP2:
	UF : 1, UT : 1,
	J1=    90.000 deg,	J2=  -100.000 deg
};
P[439]{
   GP1:
	UF : 1, UT : 1,		CONFIG : 'N U T, 0, 0, 0',
	X =  2524.463  mm,	Y =  -197.098  mm,	Z =   128.768  mm,
	W =    34.356 deg,	P =   -21.215 deg,	R =    72.687 deg
   GP2:
	UF : 1, UT : 1,
	J1=    90.000 deg,	J2=  -100.000 deg
};
P[440]{
   GP1:
	UF : 1, UT : 1,		CONFIG : 'N U T, 0, 0, 0',
	X =  2510.751  mm,	Y =   -83.956  mm,	Z =    69.338  mm,
	W =    37.818 deg,	P =   -13.036 deg,	R =    74.756 deg
   GP2:
	UF : 1, UT : 1,
	J1=    90.000 deg,	J2=  -100.000 deg
};
P[441]{
   GP1:
	UF : 1, UT : 1,		CONFIG : 'N U T, 0, 0, 0',
	X =  2526.277  mm,	Y =    63.365  mm,	Z =     6.956  mm,
	W =   -19.934 deg,	P =   -29.387 deg,	R =   -57.880 deg
   GP2:
	UF : 1, UT : 1,
	J1=    90.000 deg,	J2=   100.000 deg
};
P[442]{
   GP1:
	UF : 1, UT : 1,		CONFIG : 'N U T, 0, 0, 0',
	X =  2476.260  mm,	Y =    64.731  mm,	Z =     8.361  mm,
	W =   -19.934 deg,	P =   -29.387 deg,	R =   -63.550 deg
   GP2:
	UF : 1, UT : 1,
	J1=    90.000 deg,	J2=   100.000 deg
};
P[443]{
   GP1:
	UF : 1, UT : 1,		CONFIG : 'N U T, 0, 0, 0',
	X =  2476.548  mm,	Y =  -100.813  mm,	Z =    49.189  mm,
	W =    17.695 deg,	P =    34.286 deg,	R =    43.595 deg
   GP2:
	UF : 1, UT : 1,
	J1=    90.000 deg,	J2=  -100.000 deg
};
P[444]{
   GP1:
	UF : 1, UT : 1,		CONFIG : 'N U T, 0, 0, 0',
	X =  2544.628  mm,	Y =   -45.109  mm,	Z =    73.600  mm,
	W =     4.103 deg,	P =   -36.188 deg,	R =    83.315 deg
   GP2:
	UF : 1, UT : 1,
	J1=    90.000 deg,	J2=   -90.000 deg
};
P[445]{
   GP1:
	UF : 1, UT : 1,		CONFIG : 'N U T, 0, 0, 0',
	X =  2455.658  mm,	Y =    67.026  mm,	Z =    12.574  mm,
	W =   -19.934 deg,	P =   -29.387 deg,	R =   -80.749 deg
   GP2:
	UF : 1, UT : 1,
	J1=    90.000 deg,	J2=   100.000 deg
};
P[446]{
   GP1:
	UF : 1, UT : 1,		CONFIG : 'N U T, 0, 0, 0',
	X =  2355.398  mm,	Y =    63.665  mm,	Z =     4.813  mm,
	W =   -34.842 deg,	P =    -3.506 deg,	R =     3.705 deg
   GP2:
	UF : 1, UT : 1,
	J1=    90.000 deg,	J2=   100.000 deg
};
P[447]{
   GP1:
	UF : 1, UT : 1,		CONFIG : 'N U T, 0, 0, 0',
	X =  2497.820  mm,	Y =   -70.192  mm,	Z =   107.198  mm,
	W =    33.062 deg,	P =   -37.223 deg,	R =    56.855 deg
   GP2:
	UF : 1, UT : 1,
	J1=    90.000 deg,	J2=   -90.000 deg
};
P[448]{
   GP1:
	UF : 1, UT : 1,		CONFIG : 'N U T, 0, 0, 0',
	X =  2497.820  mm,	Y =  -198.763  mm,	Z =   107.198  mm,
	W =    47.990 deg,	P =    -4.330 deg,	R =    17.845 deg
   GP2:
	UF : 1, UT : 1,
	J1=    90.000 deg,	J2=   -90.000 deg
};
P[449]{
   GP1:
	UF : 1, UT : 1,		CONFIG : 'N U T, 0, 0, 0',
	X =  1687.303  mm,	Y =  -198.763  mm,	Z =   107.197  mm,
	W =    47.989 deg,	P =    -4.330 deg,	R =     1.515 deg
   GP2:
	UF : 1, UT : 1,
	J1=    90.000 deg,	J2=   -90.000 deg
};
P[450]{
   GP1:
	UF : 1, UT : 1,		CONFIG : 'N U T, 0, 0, 0',
	X =  2408.228  mm,	Y =    62.808  mm,	Z =     2.884  mm,
	W =   -34.842 deg,	P =    -3.506 deg,	R =     3.705 deg
   GP2:
	UF : 1, UT : 1,
	J1=    90.000 deg,	J2=   100.000 deg
};
P[451]{
   GP1:
	UF : 1, UT : 1,		CONFIG : 'N U T, 0, 0, 0',
	X =  2427.994  mm,	Y =    64.089  mm,	Z =     5.094  mm,
	W =   -26.267 deg,	P =   -23.909 deg,	R =     6.613 deg
   GP2:
	UF : 1, UT : 1,
	J1=    90.000 deg,	J2=   100.000 deg
};
P[452]{
   GP1:
	UF : 1, UT : 1,		CONFIG : 'N U T, 0, 0, 0',
	X =  2105.146  mm,	Y =   229.217  mm,	Z =   836.625  mm,
	W =     -.930 deg,	P =    44.011 deg,	R =    86.734 deg
   GP2:
	UF : 1, UT : 1,
	J1=    90.000 deg,	J2=    90.000 deg
};
P[453]{
   GP1:
	UF : 1, UT : 1,		CONFIG : 'N U T, 0, 0, 0',
	X =  2241.610  mm,	Y =   227.738  mm,	Z =   836.136  mm,
	W =     -.934 deg,	P =    44.019 deg,	R =    86.733 deg
   GP2:
	UF : 1, UT : 1,
	J1=    90.000 deg,	J2=    90.000 deg
};
P[454]{
   GP1:
	UF : 1, UT : 1,		CONFIG : 'N U T, 0, 0, 0',
	X =  2267.618  mm,	Y =   220.907  mm,	Z =   836.227  mm,
	W =      .352 deg,	P =    45.176 deg,	R =    68.647 deg
   GP2:
	UF : 1, UT : 1,
	J1=    90.000 deg,	J2=    90.000 deg
};
P[455]{
   GP1:
	UF : 1, UT : 1,		CONFIG : 'N U T, 0, 0, 0',
	X =  2288.133  mm,	Y =   209.408  mm,	Z =   838.055  mm,
	W =      .352 deg,	P =    45.176 deg,	R =    48.726 deg
   GP2:
	UF : 1, UT : 1,
	J1=    90.000 deg,	J2=    90.000 deg
};
P[456]{
   GP1:
	UF : 1, UT : 1,		CONFIG : 'N U T, 0, 0, 0',
	X =  2639.489  mm,	Y =   -80.581  mm,	Z =   838.835  mm,
	W =   -21.961 deg,	P =    40.322 deg,	R =    22.042 deg
   GP2:
	UF : 1, UT : 1,
	J1=    90.000 deg,	J2=    90.000 deg
};
P[457]{
   GP1:
	UF : 1, UT : 1,		CONFIG : 'N U T, 0, 0, 0',
	X =  2671.476  mm,	Y =  -107.218  mm,	Z =   838.434  mm,
	W =   -38.802 deg,	P =    24.854 deg,	R =    -1.556 deg
   GP2:
	UF : 1, UT : 1,
	J1=    90.000 deg,	J2=    90.000 deg
};
P[458]{
   GP1:
	UF : 1, UT : 1,		CONFIG : 'N U T, 0, 0, 0',
	X =  2691.547  mm,	Y =  -123.789  mm,	Z =   838.888  mm,
	W =   -41.798 deg,	P =    18.462 deg,	R =     1.086 deg
   GP2:
	UF : 1, UT : 1,
	J1=    90.000 deg,	J2=    90.000 deg
};
P[459]{
   GP1:
	UF : 1, UT : 1,		CONFIG : 'N U T, 0, 0, 0',
	X =  2714.691  mm,	Y =  -143.146  mm,	Z =   839.288  mm,
	W =   -41.797 deg,	P =    18.462 deg,	R =    17.758 deg
   GP2:
	UF : 1, UT : 1,
	J1=    90.000 deg,	J2=    90.000 deg
};
P[460]{
   GP1:
	UF : 1, UT : 1,		CONFIG : 'N U T, 0, 0, 0',
	X =  1451.608  mm,	Y =  -200.987  mm,	Z =   183.132  mm,
	W =     1.722 deg,	P =   -44.974 deg,	R =    59.643 deg
   GP2:
	UF : 1, UT : 1,
	J1=    90.000 deg,	J2=   -90.000 deg
};
P[461]{
   GP1:
	UF : 1, UT : 1,		CONFIG : 'N U T, 0, 0, 0',
	X =  2291.608  mm,	Y =  -200.987  mm,	Z =   183.132  mm,
	W =    44.564 deg,	P =    -7.025 deg,	R =   -20.843 deg
   GP2:
	UF : 1, UT : 1,
	J1=    90.000 deg,	J2=   -90.000 deg
};
P[462]{
   GP1:
	UF : 1, UT : 1,		CONFIG : 'N U T, 0, 0, 0',
	X =  2127.396  mm,	Y =   155.322  mm,	Z =   839.805  mm,
	W =      .687 deg,	P =    43.701 deg,	R =   155.166 deg
   GP2:
	UF : 1, UT : 1,
	J1=    90.000 deg,	J2=    90.000 deg
};
P[463]{
   GP1:
	UF : 1, UT : 1,		CONFIG : 'N U T, 0, 0, 0',
	X =  2122.679  mm,	Y =   137.192  mm,	Z =   838.754  mm,
	W =      .769 deg,	P =    43.730 deg,	R =   155.231 deg
   GP2:
	UF : 1, UT : 1,
	J1=    90.000 deg,	J2=    90.000 deg
};
P[464]{
   GP1:
	UF : 1, UT : 1,		CONFIG : 'N U T, 0, 0, 0',
	X =  2291.608  mm,	Y =  -200.987  mm,	Z =   183.132  mm,
	W =    44.564 deg,	P =    -7.025 deg,	R =   -20.843 deg
   GP2:
	UF : 1, UT : 1,
	J1=    90.000 deg,	J2=   -90.000 deg
};
P[465]{
   GP1:
	UF : 1, UT : 1,		CONFIG : 'N U T, 0, 0, 0',
	X =  2291.607  mm,	Y =  -337.988  mm,	Z =   584.132  mm,
	W =      .177 deg,	P =    -3.948 deg,	R =    26.777 deg
   GP2:
	UF : 1, UT : 1,
	J1=    90.000 deg,	J2=  -135.000 deg
};
P[466]{
   GP1:
	UF : 1, UT : 1,		CONFIG : 'N U T, 0, 0, 0',
	X =  2722.663  mm,	Y =  -266.783  mm,	Z =   377.226  mm,
	W =     0.000 deg,	P =     0.000 deg,	R =    36.754 deg
   GP2:
	UF : 1, UT : 1,
	J1=    90.000 deg,	J2=  -135.000 deg
};
P[467]{
   GP1:
	UF : 1, UT : 1,		CONFIG : 'N U T, 0, 0, 0',
	X =  2093.063  mm,	Y =   125.013  mm,	Z =   838.824  mm,
	W =      .722 deg,	P =    43.766 deg,	R =    69.804 deg
   GP2:
	UF : 1, UT : 1,
	J1=    90.000 deg,	J2=    90.000 deg
};
P[468]{
   GP1:
	UF : 1, UT : 1,		CONFIG : 'N U T, 0, 0, 0',
	X =  2081.404  mm,	Y =   152.862  mm,	Z =   838.116  mm,
	W =      .593 deg,	P =    43.021 deg,	R =   -18.687 deg
   GP2:
	UF : 1, UT : 1,
	J1=    90.000 deg,	J2=    90.000 deg
};
P[469]{
   GP1:
	UF : 1, UT : 1,		CONFIG : 'N U T, 0, 0, 0',
	X =  2722.662  mm,	Y =  -266.783  mm,	Z =   377.226  mm,
	W =    -5.375 deg,	P =   -10.513 deg,	R =    27.278 deg
   GP2:
	UF : 1, UT : 1,
	J1=    90.000 deg,	J2=  -135.000 deg
};
P[470]{
   GP1:
	UF : 1, UT : 1,		CONFIG : 'N U T, 0, 0, 0',
	X =  2382.844  mm,	Y =  -377.783  mm,	Z =   377.226  mm,
	W =      .500 deg,	P =    -4.204 deg,	R =    -6.802 deg
   GP2:
	UF : 1, UT : 1,
	J1=    90.000 deg,	J2=  -135.000 deg
};
P[471]{
   GP1:
	UF : 1, UT : 1,		CONFIG : 'N U T, 0, 0, 0',
	X =  2094.019  mm,	Y =   192.771  mm,	Z =   837.215  mm,
	W =     1.460 deg,	P =    43.967 deg,	R =   -19.119 deg
   GP2:
	UF : 1, UT : 1,
	J1=    90.000 deg,	J2=    90.000 deg
};
P[472]{
   GP1:
	UF : 1, UT : 1,		CONFIG : 'N U T, 0, 0, 0',
	X =  2121.115  mm,	Y =   201.424  mm,	Z =   840.005  mm,
	W =      .553 deg,	P =    43.710 deg,	R =  -116.800 deg
   GP2:
	UF : 1, UT : 1,
	J1=    90.000 deg,	J2=    90.000 deg
};
P[473]{
   GP1:
	UF : 1, UT : 1,		CONFIG : 'N U T, 0, 0, 0',
	X =  2382.844  mm,	Y =  -377.783  mm,	Z =   377.226  mm,
	W =      .500 deg,	P =    -4.204 deg,	R =    -6.802 deg
   GP2:
	UF : 1, UT : 1,
	J1=    90.000 deg,	J2=  -135.000 deg
};
P[474]{
   GP1:
	UF : 1, UT : 1,		CONFIG : 'N U T, 0, 0, 0',
	X =   731.273  mm,	Y =  -301.784  mm,	Z =   377.226  mm,
	W =   -10.136 deg,	P =    51.294 deg,	R =   -17.031 deg
   GP2:
	UF : 1, UT : 1,
	J1=    90.000 deg,	J2=  -135.000 deg
};
P[475]{
   GP1:
	UF : 1, UT : 1,		CONFIG : 'N U T, 0, 0, 0',
	X =   897.241  mm,	Y =   265.977  mm,	Z =   328.733  mm,
	W =   -15.049 deg,	P =    18.684 deg,	R =   -44.873 deg
   GP2:
	UF : 1, UT : 1,
	J1=    90.000 deg,	J2=   -90.000 deg
};
P[476]{
   GP1:
	UF : 1, UT : 1,		CONFIG : 'N U T, 0, 0, 0',
	X =  1702.715  mm,	Y =   146.217  mm,	Z =    77.226  mm,
	W =   -22.781 deg,	P =    33.614 deg,	R =   -37.184 deg
   GP2:
	UF : 1, UT : 1,
	J1=    90.000 deg,	J2=   -90.000 deg
};
P[477]{
   GP1:
	UF : 1, UT : 1,		CONFIG : 'N U T, 0, 0, -1',
	X =  2134.939  mm,	Y =   176.615  mm,	Z =   838.538  mm,
	W =     -.620 deg,	P =    43.564 deg,	R =   157.987 deg
   GP2:
	UF : 1, UT : 1,
	J1=    90.000 deg,	J2=    90.000 deg
};
P[478]{
   GP1:
	UF : 1, UT : 1,		CONFIG : 'N U T, 0, 0, -1',
	X =  2127.811  mm,	Y =   155.635  mm,	Z =   839.031  mm,
	W =    -1.408 deg,	P =    43.339 deg,	R =   157.483 deg
   GP2:
	UF : 1, UT : 1,
	J1=    90.000 deg,	J2=    90.000 deg
};
P[479]{
   GP1:
	UF : 1, UT : 1,		CONFIG : 'N U T, 0, 0, 0',
	X =  1713.805  mm,	Y =   111.978  mm,	Z =    49.291  mm,
	W =   -29.116 deg,	P =    35.962 deg,	R =    22.590 deg
   GP2:
	UF : 1, UT : 1,
	J1=    90.000 deg,	J2=   -90.000 deg
};
P[480]{
   GP1:
	UF : 1, UT : 1,		CONFIG : 'N U T, 0, 0, 0',
	X =  2094.232  mm,	Y =    19.822  mm,	Z =    16.623  mm,
	W =   -33.555 deg,	P =   -20.475 deg,	R =   113.896 deg
   GP2:
	UF : 1, UT : 1,
	J1=    80.000 deg,	J2=    90.000 deg
};
P[481]{
   GP1:
	UF : 1, UT : 1,		CONFIG : 'N U T, 0, 0, 0',
	X =  2206.375  mm,	Y =   -84.206  mm,	Z =    -4.653  mm,
	W =   -33.592 deg,	P =   -20.528 deg,	R =   117.916 deg
   GP2:
	UF : 1, UT : 1,
	J1=    80.000 deg,	J2=    90.000 deg
};
P[482]{
   GP1:
	UF : 1, UT : 1,		CONFIG : 'N U T, 0, 0, 0',
	X =  2255.454  mm,	Y =  -121.848  mm,	Z =   -10.027  mm,
	W =   -17.164 deg,	P =   -39.269 deg,	R =    90.811 deg
   GP2:
	UF : 1, UT : 1,
	J1=    80.000 deg,	J2=    90.000 deg
};
P[483]{
   GP1:
	UF : 1, UT : 1,		CONFIG : 'N U T, 0, 0, 0',
	X =  2303.774  mm,	Y =  -139.202  mm,	Z =   -19.217  mm,
	W =   -17.185 deg,	P =   -39.290 deg,	R =    99.791 deg
   GP2:
	UF : 1, UT : 1,
	J1=    80.000 deg,	J2=    90.000 deg
};
P[484]{
   GP1:
	UF : 1, UT : 1,		CONFIG : 'N U T, 0, 0, 0',
	X =  1968.967  mm,	Y =   144.072  mm,	Z =    81.579  mm,
	W =   -36.943 deg,	P =    -2.644 deg,	R =    15.378 deg
   GP2:
	UF : 1, UT : 1,
	J1=    90.000 deg,	J2=   -90.000 deg
};
P[485]{
   GP1:
	UF : 1, UT : 1,		CONFIG : 'N U T, 0, 0, 0',
	X =  2324.967  mm,	Y =    69.072  mm,	Z =    40.981  mm,
	W =   -36.311 deg,	P =    -7.792 deg,	R =     8.435 deg
   GP2:
	UF : 1, UT : 1,
	J1=    90.000 deg,	J2=   -90.000 deg
};
P[486]{
   GP1:
	UF : 1, UT : 1,		CONFIG : 'N U T, 0, 0, 0',
	X =  2319.749  mm,	Y =  -144.824  mm,	Z =   -20.315  mm,
	W =   -25.651 deg,	P =   -34.890 deg,	R =    98.088 deg
   GP2:
	UF : 1, UT : 1,
	J1=    80.000 deg,	J2=    90.000 deg
};
P[487]{
   GP1:
	UF : 1, UT : 1,		CONFIG : 'N U T, 0, 0, 0',
	X =  2336.580  mm,	Y =  -147.632  mm,	Z =   -22.463  mm,
	W =   -25.652 deg,	P =   -34.890 deg,	R =    87.210 deg
   GP2:
	UF : 1, UT : 1,
	J1=    80.000 deg,	J2=    90.000 deg
};
P[488]{
   GP1:
	UF : 1, UT : 1,		CONFIG : 'N U T, 0, 0, 0',
	X =  2324.967  mm,	Y =    69.072  mm,	Z =    40.981  mm,
	W =   -36.311 deg,	P =    -7.792 deg,	R =     8.435 deg
   GP2:
	UF : 1, UT : 1,
	J1=    90.000 deg,	J2=   -90.000 deg
};
P[489]{
   GP1:
	UF : 1, UT : 1,		CONFIG : 'N U T, 0, 0, 0',
	X =  2351.123  mm,	Y =   -55.973  mm,	Z =    40.981  mm,
	W =   -34.833 deg,	P =   -13.430 deg,	R =      .429 deg
   GP2:
	UF : 1, UT : 1,
	J1=    90.000 deg,	J2=   -90.000 deg
};
P[490]{
   GP1:
	UF : 1, UT : 1,		CONFIG : 'N U T, 0, 0, 0',
	X =  2111.220  mm,	Y =    30.146  mm,	Z =    16.113  mm,
	W =    23.413 deg,	P =   -33.667 deg,	R =   -79.616 deg
   GP2:
	UF : 1, UT : 1,
	J1=    80.000 deg,	J2=   -90.000 deg
};
P[491]{
   GP1:
	UF : 1, UT : 1,		CONFIG : 'N U T, 0, 0, 0',
	X =  2117.747  mm,	Y =    34.877  mm,	Z =    15.620  mm,
	W =    21.330 deg,	P =   -32.904 deg,	R =   -59.466 deg
   GP2:
	UF : 1, UT : 1,
	J1=    80.000 deg,	J2=   -90.000 deg
};
P[492]{
   GP1:
	UF : 1, UT : 1,		CONFIG : 'N U T, 0, 0, 0',
	X =  2374.335  mm,	Y =   -24.017  mm,	Z =    48.385  mm,
	W =   -44.695 deg,	P =    -5.891 deg,	R =    15.397 deg
   GP2:
	UF : 1, UT : 1,
	J1=    90.000 deg,	J2=   -90.000 deg
};
P[493]{
   GP1:
	UF : 1, UT : 1,		CONFIG : 'N U T, 0, 0, 0',
	X =  2142.335  mm,	Y =   175.983  mm,	Z =   148.385  mm,
	W =   -44.695 deg,	P =    -5.891 deg,	R =    15.397 deg
   GP2:
	UF : 1, UT : 1,
	J1=    90.000 deg,	J2=   -90.000 deg
};
P[494]{
   GP1:
	UF : 1, UT : 1,		CONFIG : 'N U T, 0, 0, 0',
	X =  1218.335  mm,	Y =   175.983  mm,	Z =   148.385  mm,
	W =   -44.695 deg,	P =    -5.891 deg,	R =    15.397 deg
   GP2:
	UF : 1, UT : 1,
	J1=    90.000 deg,	J2=   -90.000 deg
};
P[495]{
   GP1:
	UF : 1, UT : 1,		CONFIG : 'N U T, 0, 0, 0',
	X =  1218.335  mm,	Y =  -367.017  mm,	Z =  1248.385  mm,
	W =   -44.695 deg,	P =    -5.891 deg,	R =    15.397 deg
   GP2:
	UF : 1, UT : 1,
	J1=    90.000 deg,	J2=   -90.000 deg
};
P[496]{
   GP1:
	UF : 1, UT : 1,		CONFIG : 'N U T, 0, 0, 0',
	X =  2165.335  mm,	Y =  -107.803  mm,	Z =  1248.384  mm,
	W =    46.924 deg,	P =   -15.313 deg,	R =    -6.108 deg
   GP2:
	UF : 0, UT : 1,
	J1=    90.000 deg,	J2=   -90.000 deg
};
P[497]{
   GP1:
	UF : 1, UT : 1,		CONFIG : 'N U T, 0, 0, 0',
	X =  2340.715  mm,	Y =     7.886  mm,	Z =   987.384  mm,
	W =    41.825 deg,	P =    27.874 deg,	R =   -28.664 deg
   GP2:
	UF : 0, UT : 1,
	J1=    90.000 deg,	J2=   -90.000 deg
};
P[498]{
   GP1:
	UF : 1, UT : 1,		CONFIG : 'N U T, 0, 0, 0',
	X =  2116.413  mm,	Y =    35.427  mm,	Z =    15.101  mm,
	W =    12.618 deg,	P =   -40.111 deg,	R =  -122.067 deg
   GP2:
	UF : 1, UT : 1,
	J1=    79.999 deg,	J2=   -90.000 deg
};
P[499]{
   GP1:
	UF : 1, UT : 1,		CONFIG : 'N U T, 0, 0, 0',
	X =  2130.313  mm,	Y =    43.358  mm,	Z =    11.053  mm,
	W =    12.036 deg,	P =   -37.618 deg,	R =  -104.116 deg
   GP2:
	UF : 1, UT : 1,
	J1=    80.000 deg,	J2=   -90.000 deg
};
P[500]{
   GP1:
	UF : 1, UT : 1,		CONFIG : 'N U T, 0, 0, 0',
	X =  2410.122  mm,	Y =   -61.241  mm,	Z =   951.399  mm,
	W =    37.791 deg,	P =    26.519 deg,	R =   -29.934 deg
   GP2:
	UF : 0, UT : 1,
	J1=    90.000 deg,	J2=   -90.000 deg
};
P[501]{
   GP1:
	UF : 1, UT : 1,		CONFIG : 'N U T, 0, 0, 0',
	X =  2446.428  mm,	Y =    27.759  mm,	Z =   951.399  mm,
	W =    19.638 deg,	P =    41.342 deg,	R =    20.588 deg
   GP2:
	UF : 0, UT : 1,
	J1=    90.000 deg,	J2=   -90.000 deg
};
P[502]{
   GP1:
	UF : 1, UT : 1,		CONFIG : 'N U T, 0, 0, 0',
	X =  2149.942  mm,	Y =    55.888  mm,	Z =     9.504  mm,
	W =    12.076 deg,	P =   -37.629 deg,	R =   -82.652 deg
   GP2:
	UF : 1, UT : 1,
	J1=    80.000 deg,	J2=   -90.000 deg
};
P[503]{
   GP1:
	UF : 1, UT : 1,		CONFIG : 'N U T, 0, 0, 0',
	X =  2223.889  mm,	Y =   102.740  mm,	Z =    -4.406  mm,
	W =    13.123 deg,	P =   -36.448 deg,	R =   -87.052 deg
   GP2:
	UF : 1, UT : 1,
	J1=    80.000 deg,	J2=   -90.000 deg
};
P[504]{
   GP1:
	UF : 1, UT : 1,		CONFIG : 'N U T, 0, 0, 0',
	X =  2446.428  mm,	Y =    27.759  mm,	Z =   951.399  mm,
	W =    19.638 deg,	P =    41.342 deg,	R =    20.588 deg
   GP2:
	UF : 0, UT : 1,
	J1=    90.000 deg,	J2=   -90.000 deg
};
P[505]{
   GP1:
	UF : 1, UT : 1,		CONFIG : 'N U T, 0, 0, 0',
	X =  1091.922  mm,	Y =  -116.142  mm,	Z =  1409.503  mm,
	W =    -3.282 deg,	P =    29.924 deg,	R =   -13.595 deg
   GP2:
	UF : 0, UT : 1,
	J1=    90.000 deg,	J2=   -90.000 deg
};
P[506]{
   GP1:
	UF : 1, UT : 1,		CONFIG : 'N U T, 0, 0, 0',
	X =  1277.439  mm,	Y =  -574.806  mm,	Z =   798.059  mm,
	W =    19.888 deg,	P =    17.890 deg,	R =    65.874 deg
   GP2:
	UF : 1, UT : 1,
	J1=    90.000 deg,	J2=  -100.000 deg
};
P[507]{
   GP1:
	UF : 1, UT : 1,		CONFIG : 'N U T, 0, 0, 0',
	X =  1662.318  mm,	Y =  -290.218  mm,	Z =   298.449  mm,
	W =    46.284 deg,	P =    -3.804 deg,	R =    76.744 deg
   GP2:
	UF : 1, UT : 1,
	J1=    90.000 deg,	J2=  -100.000 deg
};
P[508]{
   GP1:
	UF : 1, UT : 1,		CONFIG : 'N U T, 0, 0, 0',
	X =  2054.473  mm,	Y =  -224.770  mm,	Z =   280.594  mm,
	W =    49.761 deg,	P =   -15.389 deg,	R =    77.321 deg
   GP2:
	UF : 1, UT : 1,
	J1=    90.000 deg,	J2=  -100.000 deg
};
P[509]{
   GP1:
	UF : 1, UT : 1,		CONFIG : 'N U T, 0, 0, 0',
	X =  2054.474  mm,	Y =   -24.769  mm,	Z =   118.594  mm,
	W =    48.014 deg,	P =    21.400 deg,	R =    69.846 deg
   GP2:
	UF : 1, UT : 1,
	J1=    90.000 deg,	J2=  -100.000 deg
};
P[510]{
   GP1:
	UF : 1, UT : 1,		CONFIG : 'N U T, 0, 0, 0',
	X =  2256.562  mm,	Y =   119.443  mm,	Z =    -9.324  mm,
	W =     8.564 deg,	P =   -38.851 deg,	R =   -87.708 deg
   GP2:
	UF : 1, UT : 1,
	J1=    80.000 deg,	J2=   -90.000 deg
};
P[511]{
   GP1:
	UF : 1, UT : 1,		CONFIG : 'N U T, 0, 0, 0',
	X =  2298.877  mm,	Y =   133.398  mm,	Z =   -15.964  mm,
	W =   -25.455 deg,	P =   -35.130 deg,	R =   -43.698 deg
   GP2:
	UF : 1, UT : 1,
	J1=    80.000 deg,	J2=   -90.000 deg
};
P[512]{
   GP1:
	UF : 1, UT : 1,		CONFIG : 'N U T, 0, 0, 0',
	X =  2054.474  mm,	Y =   -24.769  mm,	Z =   118.594  mm,
	W =    48.014 deg,	P =    21.400 deg,	R =    69.846 deg
   GP2:
	UF : 1, UT : 1,
	J1=    90.000 deg,	J2=  -100.000 deg
};
P[513]{
   GP1:
	UF : 1, UT : 1,		CONFIG : 'N U T, 0, 0, 0',
	X =  2210.473  mm,	Y =  -152.769  mm,	Z =   150.477  mm,
	W =    50.237 deg,	P =    13.157 deg,	R =   -13.726 deg
   GP2:
	UF : 1, UT : 1,
	J1=    90.000 deg,	J2=   -90.000 deg
};
P[514]{
   GP1:
	UF : 1, UT : 1,		CONFIG : 'N U T, 0, 0, 0',
	X =  2551.972  mm,	Y =  -676.778  mm,	Z =   -60.803  mm,
	W =   -25.914 deg,	P =   -20.730 deg,	R =    53.931 deg
   GP2:
	UF : 1, UT : 1,
	J1=    80.000 deg,	J2=    90.000 deg
};
P[515]{
   GP1:
	UF : 1, UT : 1,		CONFIG : 'N U T, 0, 0, 0',
	X =  2554.061  mm,	Y =  -660.992  mm,	Z =   -63.273  mm,
	W =   -25.035 deg,	P =   -20.126 deg,	R =    53.624 deg
   GP2:
	UF : 1, UT : 1,
	J1=    80.000 deg,	J2=    90.000 deg
};
P[516]{
   GP1:
	UF : 1, UT : 1,		CONFIG : 'N U T, 0, 0, 0',
	X =  2223.625  mm,	Y =   -98.572  mm,	Z =    36.411  mm,
	W =    43.410 deg,	P =    13.252 deg,	R =   -13.621 deg
   GP2:
	UF : 1, UT : 1,
	J1=    90.000 deg,	J2=   -90.000 deg
};
P[517]{
   GP1:
	UF : 1, UT : 1,		CONFIG : 'N U T, 0, 0, 0',
	X =  2555.644  mm,	Y =  -656.185  mm,	Z =   -64.155  mm,
	W =   -33.504 deg,	P =     -.369 deg,	R =    59.795 deg
   GP2:
	UF : 1, UT : 1,
	J1=    80.000 deg,	J2=    90.000 deg
};
P[518]{
   GP1:
	UF : 1, UT : 1,		CONFIG : 'N U T, 0, 0, 1',
	X =  2567.112  mm,	Y =  -646.430  mm,	Z =   -62.505  mm,
	W =   -33.129 deg,	P =   -11.990 deg,	R =    19.464 deg
   GP2:
	UF : 1, UT : 1,
	J1=    80.000 deg,	J2=    90.000 deg
};
P[519]{
   GP1:
	UF : 1, UT : 1,		CONFIG : 'N U T, 0, 0, 0',
	X =  1989.335  mm,	Y =   -96.402  mm,	Z =    22.227  mm,
	W =    43.411 deg,	P =    13.252 deg,	R =   -13.621 deg
   GP2:
	UF : 1, UT : 1,
	J1=    90.000 deg,	J2=   -90.000 deg
};
P[520]{
   GP1:
	UF : 1, UT : 1,		CONFIG : 'N U T, 0, 0, 0',
	X =  2615.881  mm,	Y =  -607.927  mm,	Z =   -73.286  mm,
	W =   -31.218 deg,	P =    -7.950 deg,	R =    48.121 deg
   GP2:
	UF : 1, UT : 1,
	J1=    80.000 deg,	J2=    90.000 deg
};
P[521]{
   GP1:
	UF : 1, UT : 1,		CONFIG : 'N U T, 0, 0, 0',
	X =  2626.109  mm,	Y =  -566.903  mm,	Z =   -73.840  mm,
	W =   -26.872 deg,	P =   -18.421 deg,	R =    63.003 deg
   GP2:
	UF : 1, UT : 1,
	J1=    80.000 deg,	J2=    90.000 deg
};
P[522]{
   GP1:
	UF : 1, UT : 1,		CONFIG : 'N U T, 0, 0, 0',
	X =  2496.861  mm,	Y =  -851.474  mm,	Z =     -.087  mm,
	W =   -43.356 deg,	P =    13.468 deg,	R =   106.076 deg
   GP2:
	UF : 1, UT : 1,
	J1=    90.000 deg,	J2=   -90.000 deg
};
P[523]{
   GP1:
	UF : 1, UT : 1,		CONFIG : 'N U T, 0, 0, 0',
	X =  2058.051  mm,	Y =  -175.228  mm,	Z =   206.322  mm,
	W =    46.132 deg,	P =   -12.958 deg,	R =   -13.413 deg
   GP2:
	UF : 1, UT : 1,
	J1=    90.000 deg,	J2=   -90.000 deg
};
P[524]{
   GP1:
	UF : 1, UT : 1,		CONFIG : 'N U T, 0, 0, 0',
	X =  1948.050  mm,	Y =  -251.228  mm,	Z =   206.322  mm,
	W =   -42.705 deg,	P =    -6.373 deg,	R =    58.147 deg
   GP2:
	UF : 1, UT : 1,
	J1=    90.000 deg,	J2=   -90.000 deg
};
P[525]{
   GP1:
	UF : 1, UT : 1,		CONFIG : 'N U T, 0, 0, 0',
	X =  1948.050  mm,	Y =  -151.228  mm,	Z =    88.322  mm,
	W =   -42.016 deg,	P =    10.583 deg,	R =    76.528 deg
   GP2:
	UF : 1, UT : 1,
	J1=    90.000 deg,	J2=   -90.000 deg
};
P[526]{
   GP1:
	UF : 1, UT : 1,		CONFIG : 'N U T, 0, 0, 0',
	X =  2494.766  mm,	Y =  -783.515  mm,	Z =     1.726  mm,
	W =   -43.359 deg,	P =    13.457 deg,	R =   106.066 deg
   GP2:
	UF : 1, UT : 1,
	J1=    90.000 deg,	J2=   -90.000 deg
};
P[527]{
   GP1:
	UF : 1, UT : 1,		CONFIG : 'N U T, 0, 0, 0',
	X =  2518.465  mm,	Y =  -758.192  mm,	Z =     -.116  mm,
	W =   -37.799 deg,	P =   -26.510 deg,	R =   -29.925 deg
   GP2:
	UF : 1, UT : 1,
	J1=    90.000 deg,	J2=   -90.000 deg
};
P[528]{
   GP1:
	UF : 1, UT : 1,		CONFIG : 'N U T, 0, 0, 1',
	X =  1919.292  mm,	Y =  -155.329  mm,	Z =    58.531  mm,
	W =   -29.954 deg,	P =    35.300 deg,	R =   158.688 deg
   GP2:
	UF : 1, UT : 1,
	J1=    90.000 deg,	J2=   -90.000 deg
};
P[529]{
   GP1:
	UF : 1, UT : 1,		CONFIG : 'N U T, 0, 0, 0',
	X =  1284.066  mm,	Y =  -721.135  mm,	Z =    74.949  mm,
	W =   -12.631 deg,	P =    46.016 deg,	R =    -5.788 deg
   GP2:
	UF : 1, UT : 1,
	J1=    90.000 deg,	J2=   -90.000 deg
};
P[530]{
   GP1:
	UF : 1, UT : 1,		CONFIG : 'N U T, 0, 0, 0',
	X =  1387.863  mm,	Y =  -282.758  mm,	Z =  1218.271  mm,
	W =      .355 deg,	P =    36.366 deg,	R =   -97.933 deg
   GP2:
	UF : 1, UT : 1,
	J1=    90.000 deg,	J2=   -90.000 deg
};
P[531]{
   GP1:
	UF : 1, UT : 1,		CONFIG : 'N U T, 0, 0, 0',
	X =  2131.864  mm,	Y =  -267.378  mm,	Z =   958.286  mm,
	W =      .355 deg,	P =    36.366 deg,	R =   -97.933 deg
   GP2:
	UF : 1, UT : 1,
	J1=    90.000 deg,	J2=   -90.000 deg
};
P[532]{
   GP1:
	UF : 1, UT : 1,		CONFIG : 'N U T, 0, 0, 0',
	X =  2564.966  mm,	Y =  -757.763  mm,	Z =      .954  mm,
	W =   -37.799 deg,	P =   -26.510 deg,	R =   -29.925 deg
   GP2:
	UF : 1, UT : 1,
	J1=    90.000 deg,	J2=   -90.000 deg
};
P[533]{
   GP1:
	UF : 1, UT : 1,		CONFIG : 'N U T, 0, 0, 0',
	X =  2439.719  mm,	Y =   -63.381  mm,	Z =     7.737  mm,
	W =    37.820 deg,	P =   -13.031 deg,	R =    74.753 deg
   GP2:
	UF : 1, UT : 1,
	J1=    90.000 deg,	J2=  -100.000 deg
};
P[534]{
   GP1:
	UF : 1, UT : 1,		CONFIG : 'N U T, 0, 0, 0',
	X =  2438.182  mm,	Y =   -87.880  mm,	Z =     8.378  mm,
	W =    36.507 deg,	P =    16.766 deg,	R =    81.655 deg
   GP2:
	UF : 1, UT : 1,
	J1=    90.000 deg,	J2=  -100.000 deg
};
P[535]{
   GP1:
	UF : 1, UT : 1,		CONFIG : 'N U T, 0, 0, 0',
	X =  2439.037  mm,	Y =  -126.347  mm,	Z =    16.024  mm,
	W =    36.512 deg,	P =    16.766 deg,	R =    82.316 deg
   GP2:
	UF : 1, UT : 1,
	J1=    90.000 deg,	J2=  -100.000 deg
};
P[536]{
   GP1:
	UF : 1, UT : 1,		CONFIG : 'N U T, 0, 0, 0',
	X =  2439.331  mm,	Y =  -141.407  mm,	Z =    20.177  mm,
	W =    33.075 deg,	P =    28.111 deg,	R =    91.096 deg
   GP2:
	UF : 1, UT : 1,
	J1=    90.000 deg,	J2=  -100.000 deg
};
P[537]{
   GP1:
	UF : 1, UT : 1,		CONFIG : 'N U T, 0, 0, 0',
	X =  2504.883  mm,	Y =    10.258  mm,	Z =     4.530  mm,
	W =    15.432 deg,	P =   -38.749 deg,	R =    78.167 deg
   GP2:
	UF : 1, UT : 1,
	J1=    90.000 deg,	J2=   -90.000 deg
};
P[538]{
   GP1:
	UF : 1, UT : 1,		CONFIG : 'N U T, 0, 0, 0',
	X =  2682.606  mm,	Y =    41.024  mm,	Z =   922.793  mm,
	W =    34.567 deg,	P =    32.862 deg,	R =   -60.440 deg
   GP2:
	UF : 1, UT : 1,
	J1=    90.000 deg,	J2=   -90.000 deg
};
P[539]{
   GP1:
	UF : 1, UT : 1,		CONFIG : 'N U T, 0, 0, 0',
	X =  2091.653  mm,	Y =  -160.976  mm,	Z =   922.793  mm,
	W =    -5.705 deg,	P =    39.927 deg,	R =  -167.749 deg
   GP2:
	UF : 1, UT : 1,
	J1=    90.000 deg,	J2=   -90.000 deg
};
P[540]{
   GP1:
	UF : 1, UT : 1,		CONFIG : 'N U T, 0, 0, 0',
	X =  2452.621  mm,	Y =    11.213  mm,	Z =     3.541  mm,
	W =    15.421 deg,	P =   -38.793 deg,	R =    78.144 deg
   GP2:
	UF : 1, UT : 1,
	J1=    90.000 deg,	J2=   -90.000 deg
};
P[541]{
   GP1:
	UF : 1, UT : 1,		CONFIG : 'N U T, 0, 0, 0',
	X =  2443.542  mm,	Y =    10.715  mm,	Z =     4.572  mm,
	W =    15.421 deg,	P =   -38.793 deg,	R =    92.357 deg
   GP2:
	UF : 1, UT : 1,
	J1=    90.000 deg,	J2=   -90.000 deg
};
P[542]{
   GP1:
	UF : 1, UT : 1,		CONFIG : 'N U T, 0, 0, 0',
	X =  1688.136  mm,	Y =   -62.029  mm,	Z =   -11.830  mm,
	W =    44.899 deg,	P =    -2.949 deg,	R =     6.765 deg
   GP2:
	UF : 1, UT : 1,
	J1=    90.000 deg,	J2=   -90.000 deg
};
P[543]{
   GP1:
	UF : 1, UT : 1,		CONFIG : 'N U T, 0, 0, 0',
	X =  1649.697  mm,	Y =   -61.920  mm,	Z =   -11.739  mm,
	W =    44.923 deg,	P =    -2.958 deg,	R =     5.948 deg
   GP2:
	UF : 1, UT : 1,
	J1=    90.000 deg,	J2=   -90.000 deg
};
P[544]{
   GP1:
	UF : 1, UT : 1,		CONFIG : 'N U T, 0, 0, 0',
	X =  1638.071  mm,	Y =   -63.852  mm,	Z =   -13.382  mm,
	W =    44.923 deg,	P =    -2.958 deg,	R =    30.934 deg
   GP2:
	UF : 1, UT : 1,
	J1=    90.000 deg,	J2=   -90.000 deg
};
P[545]{
   GP1:
	UF : 1, UT : 1,		CONFIG : 'N U T, 0, 0, 0',
	X =  1631.622  mm,	Y =   -70.088  mm,	Z =   -12.380  mm,
	W =    44.727 deg,	P =     5.577 deg,	R =    39.396 deg
   GP2:
	UF : 1, UT : 1,
	J1=    90.000 deg,	J2=   -90.000 deg
};
P[546]{
   GP1:
	UF : 1, UT : 1,		CONFIG : 'N U T, 0, 0, 0',
	X =  1604.527  mm,	Y =   -99.847  mm,	Z =   -10.764  mm,
	W =    44.727 deg,	P =     5.577 deg,	R =    41.589 deg
   GP2:
	UF : 1, UT : 1,
	J1=    90.000 deg,	J2=   -90.000 deg
};
P[547]{
   GP1:
	UF : 1, UT : 1,		CONFIG : 'N U T, 0, 0, 1',
	X =  1865.403  mm,	Y =  -247.947  mm,	Z =  1181.723  mm,
	W =   -12.320 deg,	P =    37.383 deg,	R =  -179.360 deg
   GP2:
	UF : 1, UT : 1,
	J1=    90.000 deg,	J2=   -90.000 deg
};
P[548]{
   GP1:
	UF : 1, UT : 1,		CONFIG : 'N U T, 0, 0, 0',
	X =   732.832  mm,	Y =   236.053  mm,	Z =  1006.723  mm,
	W =   -38.649 deg,	P =     6.276 deg,	R =    12.974 deg
   GP2:
	UF : 1, UT : 1,
	J1=    90.000 deg,	J2=   -90.000 deg
};
P[549]{
   GP1:
	UF : 1, UT : 1,		CONFIG : 'N U T, 0, 0, 0',
	X =  1743.832  mm,	Y =   113.053  mm,	Z =   141.722  mm,
	W =   -44.065 deg,	P =    11.483 deg,	R =   -10.762 deg
   GP2:
	UF : 1, UT : 1,
	J1=    90.000 deg,	J2=   -90.000 deg
};
P[550]{
   GP1:
	UF : 1, UT : 1,		CONFIG : 'N U T, 0, 0, 0',
	X =  1579.711  mm,	Y =  -108.035  mm,	Z =   -10.500  mm,
	W =    39.341 deg,	P =   -22.846 deg,	R =    22.246 deg
   GP2:
	UF : 1, UT : 1,
	J1=    90.000 deg,	J2=   -90.000 deg
};
P[551]{
   GP1:
	UF : 1, UT : 1,		CONFIG : 'N U T, 0, 0, 0',
	X =  1561.920  mm,	Y =   -83.236  mm,	Z =    -9.721  mm,
	W =   -23.520 deg,	P =   -39.540 deg,	R =    41.279 deg
   GP2:
	UF : 1, UT : 1,
	J1=    90.000 deg,	J2=   -90.000 deg
};
P[552]{
   GP1:
	UF : 1, UT : 1,		CONFIG : 'N U T, 0, 0, 0',
	X =  1558.907  mm,	Y =   -36.151  mm,	Z =   -10.999  mm,
	W =   -25.567 deg,	P =   -38.384 deg,	R =    42.613 deg
   GP2:
	UF : 1, UT : 1,
	J1=    90.000 deg,	J2=   -90.000 deg
};
P[553]{
   GP1:
	UF : 1, UT : 1,		CONFIG : 'N U T, 0, 0, 0',
	X =  1950.533  mm,	Y =    42.756  mm,	Z =   152.316  mm,
	W =   -44.065 deg,	P =    11.483 deg,	R =    13.279 deg
   GP2:
	UF : 1, UT : 1,
	J1=    90.000 deg,	J2=   -90.000 deg
};
P[554]{
   GP1:
	UF : 1, UT : 1,		CONFIG : 'N U T, 0, 0, 0',
	X =  2150.533  mm,	Y =    42.756  mm,	Z =    86.316  mm,
	W =   -44.065 deg,	P =    11.483 deg,	R =    13.279 deg
   GP2:
	UF : 1, UT : 1,
	J1=    90.000 deg,	J2=   -90.000 deg
};
P[555]{
   GP1:
	UF : 1, UT : 1,		CONFIG : 'N U T, 0, 0, 0',
	X =  1554.651  mm,	Y =   -28.866  mm,	Z =   -10.539  mm,
	W =   -23.520 deg,	P =   -39.540 deg,	R =    72.199 deg
   GP2:
	UF : 1, UT : 1,
	J1=    90.000 deg,	J2=   -90.000 deg
};
P[556]{
   GP1:
	UF : 1, UT : 1,		CONFIG : 'N U T, 0, 0, 0',
	X =  1541.060  mm,	Y =   -26.299  mm,	Z =   -11.935  mm,
	W =   -23.653 deg,	P =   -40.441 deg,	R =   108.581 deg
   GP2:
	UF : 1, UT : 1,
	J1=    90.000 deg,	J2=   -90.000 deg
};
P[557]{
   GP1:
	UF : 1, UT : 1,		CONFIG : 'N U T, 0, 0, 0',
	X =  2190.699  mm,	Y =   -15.223  mm,	Z =    38.789  mm,
	W =   -43.651 deg,	P =    12.243 deg,	R =    12.532 deg
   GP2:
	UF : 1, UT : 1,
	J1=    90.000 deg,	J2=   -90.000 deg
};
P[558]{
   GP1:
	UF : 1, UT : 1,		CONFIG : 'N U T, 0, 0, 0',
	X =  2364.471  mm,	Y =    13.944  mm,	Z =     1.114  mm,
	W =    44.968 deg,	P =     1.925 deg,	R =    -1.926 deg
   GP2:
	UF : 1, UT : 1,
	J1=    90.000 deg,	J2=   -90.000 deg
};
P[559]{
   GP1:
	UF : 1, UT : 1,		CONFIG : 'N U T, 0, 0, 0',
	X =  2401.563  mm,	Y =    16.505  mm,	Z =      .800  mm,
	W =    44.555 deg,	P =    -6.719 deg,	R =    -4.136 deg
   GP2:
	UF : 1, UT : 1,
	J1=    89.999 deg,	J2=   -90.000 deg
};
P[560]{
   GP1:
	UF : 1, UT : 1,		CONFIG : 'N U T, 0, 0, 0',
	X =  2095.142  mm,	Y =    -6.873  mm,	Z =    39.768  mm,
	W =   -46.048 deg,	P =     1.387 deg,	R =    -1.362 deg
   GP2:
	UF : 1, UT : 1,
	J1=    90.000 deg,	J2=   -90.000 deg
};
P[561]{
   GP1:
	UF : 1, UT : 1,		CONFIG : 'N U T, 0, 0, 0',
	X =  2427.641  mm,	Y =    15.325  mm,	Z =     3.488  mm,
	W =    36.323 deg,	P =   -28.640 deg,	R =     -.319 deg
   GP2:
	UF : 1, UT : 1,
	J1=    90.000 deg,	J2=   -90.000 deg
};
P[562]{
   GP1:
	UF : 1, UT : 1,		CONFIG : 'N U T, 0, 0, 0',
	X =  2756.905  mm,	Y =  -263.426  mm,	Z =   282.139  mm,
	W =     -.001 deg,	P =      .004 deg,	R =    26.800 deg
   GP2:
	UF : 1, UT : 1,
	J1=    90.000 deg,	J2=  -135.000 deg
};
P[563]{
   GP1:
	UF : 1, UT : 1,		CONFIG : 'N U T, 0, 0, 0',
	X =  2059.854  mm,	Y =   139.575  mm,	Z =   116.497  mm,
	W =   -43.126 deg,	P =    18.070 deg,	R =     3.079 deg
   GP2:
	UF : 1, UT : 1,
	J1=    90.000 deg,	J2=   -90.000 deg
};
P[564]{
   GP1:
	UF : 1, UT : 1,		CONFIG : 'N U T, 0, 0, 0',
	X =  2867.649  mm,	Y =  -263.060  mm,	Z =   288.229  mm,
	W =   -12.814 deg,	P =   -19.263 deg,	R =    25.759 deg
   GP2:
	UF : 1, UT : 1,
	J1=    90.000 deg,	J2=  -135.000 deg
};
P[565]{
   GP1:
	UF : 1, UT : 1,		CONFIG : 'N U T, 0, 0, 0',
	X =  1914.760  mm,	Y =  1445.095  mm,	Z =  1037.108  mm,
	W =    42.423 deg,	P =    16.662 deg,	R =   -14.263 deg
   GP2:
	UF : 1, UT : 1,
	J1=   180.000 deg,	J2=    90.000 deg
};
P[566]{
   GP1:
	UF : 1, UT : 1,		CONFIG : 'N U T, 0, 0, 0',
	X =  1597.456  mm,	Y =   176.449  mm,	Z =    24.499  mm,
	W =    17.337 deg,	P =    42.452 deg,	R =  -154.363 deg
   GP2:
	UF : 1, UT : 1,
	J1=    90.000 deg,	J2=   -90.000 deg
};
P[567]{
   GP1:
	UF : 1, UT : 1,		CONFIG : 'N U T, 0, 0, 0',
	X =  2588.510  mm,	Y =   186.120  mm,	Z =   -63.295  mm,
	W =   -40.710 deg,	P =   -12.372 deg,	R =      .282 deg
   GP2:
	UF : 1, UT : 1,
	J1=    80.000 deg,	J2=   -90.000 deg
};
P[568]{
   GP1:
	UF : 1, UT : 1,		CONFIG : 'N U T, 0, 0, 0',
	X =  2632.018  mm,	Y =   212.269  mm,	Z =   -70.671  mm,
	W =   -16.773 deg,	P =   -29.886 deg,	R =   -20.810 deg
   GP2:
	UF : 1, UT : 1,
	J1=    80.000 deg,	J2=   -90.000 deg
};
P[569]{
   GP1:
	UF : 1, UT : 1,		CONFIG : 'N U T, 0, 0, -1',
	X =  1413.425  mm,	Y =    86.564  mm,	Z =   243.315  mm,
	W =    35.973 deg,	P =    30.977 deg,	R =  -149.882 deg
   GP2:
	UF : 1, UT : 1,
	J1=    90.000 deg,	J2=   -90.000 deg
};
P[570]{
   GP1:
	UF : 1, UT : 1,		CONFIG : 'N U T, 0, 0, 0',
	X =  1396.163  mm,	Y =    95.442  mm,	Z =   229.882  mm,
	W =    36.884 deg,	P =    -6.321 deg,	R =   -64.014 deg
   GP2:
	UF : 1, UT : 1,
	J1=    80.000 deg,	J2=   -90.000 deg
};
P[571]{
   GP1:
	UF : 1, UT : 1,		CONFIG : 'N U T, 0, 0, 0',
	X =  2035.138  mm,	Y =    95.442  mm,	Z =   116.882  mm,
	W =    36.883 deg,	P =    -6.321 deg,	R =   -86.693 deg
   GP2:
	UF : 1, UT : 1,
	J1=    80.000 deg,	J2=   -90.000 deg
};
P[572]{
   GP1:
	UF : 1, UT : 1,		CONFIG : 'N U T, 0, 0, 0',
	X =  1669.539  mm,	Y =   147.286  mm,	Z =   -13.746  mm,
	W =   -26.040 deg,	P =    35.756 deg,	R =   -36.092 deg
   GP2:
	UF : 1, UT : 1,
	J1=    90.000 deg,	J2=   -90.000 deg
};
P[573]{
   GP1:
	UF : 1, UT : 1,		CONFIG : 'N U T, 0, 0, 0',
	X =  1670.050  mm,	Y =   100.399  mm,	Z =   -12.949  mm,
	W =   -26.718 deg,	P =    37.664 deg,	R =   -37.273 deg
   GP2:
	UF : 1, UT : 1,
	J1=    90.000 deg,	J2=   -90.000 deg
};
P[574]{
   GP1:
	UF : 1, UT : 1,		CONFIG : 'N U T, 0, 0, 0',
	X =  1670.267  mm,	Y =    88.409  mm,	Z =   -12.292  mm,
	W =   -26.718 deg,	P =    37.664 deg,	R =    -4.100 deg
   GP2:
	UF : 1, UT : 1,
	J1=    90.000 deg,	J2=   -90.000 deg
};
P[575]{
   GP1:
	UF : 1, UT : 1,		CONFIG : 'N U T, 0, 0, 0',
	X =  1670.710  mm,	Y =    89.750  mm,	Z =   -10.623  mm,
	W =   -33.311 deg,	P =    24.086 deg,	R =    -7.323 deg
   GP2:
	UF : 1, UT : 1,
	J1=    89.999 deg,	J2=   -90.000 deg
};
P[576]{
   GP1:
	UF : 1, UT : 1,		CONFIG : 'N U T, 0, 0, 0',
	X =  1539.625  mm,	Y = -1470.562  mm,	Z =  1075.975  mm,
	W =   -42.854 deg,	P =   -15.295 deg,	R =    39.123 deg
   GP2:
	UF : 1, UT : 1,
	J1=   180.000 deg,	J2=  -125.000 deg
};
P[577]{
   GP1:
	UF : 1, UT : 1,		CONFIG : 'N U T, 0, 0, 0',
	X =  1693.242  mm,	Y =    90.339  mm,	Z =   -10.067  mm,
	W =   -31.545 deg,	P =    22.877 deg,	R =    21.402 deg
   GP2:
	UF : 1, UT : 1,
	J1=    90.000 deg,	J2=   -90.000 deg
};
P[578]{
   GP1:
	UF : 1, UT : 1,		CONFIG : 'N U T, 0, 0, 0',
	X =  1970.669  mm,	Y =    89.152  mm,	Z =   -12.326  mm,
	W =   -33.410 deg,	P =    24.055 deg,	R =    37.165 deg
   GP2:
	UF : 1, UT : 1,
	J1=    90.000 deg,	J2=   -90.000 deg
};
P[579]{
   GP1:
	UF : 1, UT : 1,		CONFIG : 'N U T, 0, 0, 0',
	X =  1998.760  mm,	Y =    90.877  mm,	Z =    -8.459  mm,
	W =   -45.190 deg,	P =    -4.344 deg,	R =    36.475 deg
   GP2:
	UF : 1, UT : 1,
	J1=    90.000 deg,	J2=   -90.000 deg
};
P[580]{
   GP1:
	UF : 1, UT : 1,		CONFIG : 'N U T, 0, 0, 0',
	X =  2365.251  mm,	Y =    22.628  mm,	Z =    -2.109  mm,
	W =   -44.993 deg,	P =      .940 deg,	R =     6.369 deg
   GP2:
	UF : 1, UT : 1,
	J1=    90.000 deg,	J2=   -90.000 deg
};
P[581]{
   GP1:
	UF : 1, UT : 1,		CONFIG : 'N U T, 0, 0, 0',
	X =  2508.618  mm,	Y =    25.743  mm,	Z =     2.034  mm,
	W =   -44.996 deg,	P =      .946 deg,	R =     6.368 deg
   GP2:
	UF : 1, UT : 1,
	J1=    90.000 deg,	J2=   -90.000 deg
};
P[582]{
   GP1:
	UF : 1, UT : 1,		CONFIG : 'N U T, 0, 0, 0',
	X =  2363.154  mm,	Y =   -73.963  mm,	Z =     -.369  mm,
	W =   -41.235 deg,	P =    -5.523 deg,	R =     1.452 deg
   GP2:
	UF : 1, UT : 1,
	J1=    90.000 deg,	J2=   -90.000 deg
};
P[583]{
   GP1:
	UF : 1, UT : 1,		CONFIG : 'N U T, 0, 0, 0',
	X =  2405.285  mm,	Y =   -73.535  mm,	Z =     -.369  mm,
	W =   -41.235 deg,	P =    -5.523 deg,	R =     1.452 deg
   GP2:
	UF : 1, UT : 1,
	J1=    90.000 deg,	J2=   -90.000 deg
};
P[584]{
   GP1:
	UF : 1, UT : 1,		CONFIG : 'N U T, 0, 0, 0',
	X =  2428.032  mm,	Y =   -72.786  mm,	Z =     1.628  mm,
	W =   -37.657 deg,	P =   -19.014 deg,	R =    15.034 deg
   GP2:
	UF : 1, UT : 1,
	J1=    90.000 deg,	J2=   -90.000 deg
